// TwinCAT 3 PLC project Code
// ProgramVersion: 3.1.4026.25
// libraries:
//   ApplicationBase, * (Beckhoff Automation LLC)
//   Tc2_MC2, * (Beckhoff Automation GmbH)
//   Tc2_MC2_Camming, * (Beckhoff Automation GmbH)
//   Tc2_Standard, * (Beckhoff Automation GmbH)
//   Tc2_System, * (Beckhoff Automation GmbH)
//   XtsCore, * (Beckhoff Automation LLC)
// project tree:
//   / Godot.TcPOU, MAIN.TcPOU, PlcTask.TcTTO
//   POUs/ GodotHmi.TcPOU
//   Tests/Base/Interface/ I_SequenceTest.TcIO
//   Tests/CamBuild/ CamBuild.TcPOU, SplitCamBuild.TcPOU, ST_Camming.TcDUT
//   Tests/CamBuild/Interface/ I_CamBuildSequence.TcIO
//   Tests/CamCurveCompTest/ CamCurveComp.TcPOU, SplitCamRun.TcPOU, I_CamCurveComp.TcIO
//   Tests/ FB_XtsBallCamBuilder.TcPOU
// real-time tasks:
//   TASK PlcTask: cycle T#2ms, priority 20, ADS port 350
//   TASK XTS Task 1: cycle T#250us, priority 1, ADS port 351
//   TASK XTS AUX Task 1: cycle T#250us, priority 2, ADS port 352
//   TASK Job Task: cycle default, priority 32
// motion (NC):
//   TASK NC-Task 1: cycle T#2ms, priority 4, ADS port 501
//   TASK NC-Task 1 SVB: cycle T#10ms, priority 8, ADS port 511
//   AXIS Mover Axis 1 (id 1)
//     Dynamic: AccelerationMaximum=80000, DecelerationMaximum=80000, Acceleration=20000, Deceleration=20000, Jerk=200000
//     Velo: Maximum=4000
//     PositionAreaControl: Enable=false
//     TargetPosControl: Enable=false
//     OtherSettings: AllowMotionCmdToSlave=true, AllowMotionCmdToExtSetGenAxis=true
//     encoder EncType=28
//       EncPara: ModuloFactor=1500, ToleranceWndModuloStart=0.2, MaxCount=#xffffffff
//     drive DrvType=22
//       DrvPara: MaxCount=#xffffffff, DriveControlDWord=#x00000100
//         Analog: VeloReferenz=4200, TorqueSetpointScale=10
//         TimeComp: TaskDelayCycles=1
//     controller CtrType=1
//       CtrPara: PriorControlFactor=1
//         PosDiffControl: Range=75
//         Observer: BandWidth=20
//   AXIS Mover Axis 2 (id 2)
//     Dynamic: AccelerationMaximum=80000, DecelerationMaximum=80000, Acceleration=20000, Deceleration=20000, Jerk=200000
//     Velo: Maximum=4000
//     PositionAreaControl: Enable=false
//     TargetPosControl: Enable=false
//     OtherSettings: AllowMotionCmdToSlave=true, AllowMotionCmdToExtSetGenAxis=true
//     encoder EncType=28
//       EncPara: ModuloFactor=1500, ToleranceWndModuloStart=0.2, MaxCount=#xffffffff
//     drive DrvType=22
//       DrvPara: MaxCount=#xffffffff, DriveControlDWord=#x00000100
//         Analog: VeloReferenz=4200, TorqueSetpointScale=10
//         TimeComp: TaskDelayCycles=1
//     controller CtrType=1
//       CtrPara: PriorControlFactor=1
//         PosDiffControl: Range=50
//         Observer: BandWidth=20
//   AXIS VirtualMaster (id 3)
//     OtherSettings: AllowMotionCmdToSlave=true
//     encoder EncType=1
//       EncPara: ModuloFactor=1500
//     drive DrvType=5
//       Analog: TorqueSetpointScale=10, ScaleFactorActTorque=0.1
//       TimeComp: TaskDelayCycles=1
//     controller CtrType=1
//       CtrPara: PriorControlFactor=1
//         Observer: BandWidth=20
//   AXIS FeedAxis (id 4)
//     OtherSettings: AllowMotionCmdToSlave=true
//     encoder EncType=1
//     drive DrvType=5
//       Analog: TorqueSetpointScale=10, ScaleFactorActTorque=0.1
//       TimeComp: TaskDelayCycles=1
//     controller CtrType=1
//       CtrPara: PriorControlFactor=1
//         Observer: BandWidth=20
// I/O:
//   DEVICE Device 1 (EtherCAT), AmsNetId 192.168.1.107.2.1
//     Term 1 (EK1100) [EK1100 EtherCAT Coupler (2A E-Bus)]
//       Term 2 (EL1259) [EL1259 8Ch. Dig Input 24V/8Ch. Dig. Output 24V with Multi-Time-Stamp]
//       Term 3 (EL9227-5500) [EL9227-5500 Overcurrent protection 24V DC, 2Ch., max. 10A (sum), adjustable, extended functionalities]
//       Term 4 (EL9227-6644) [EL9227-6644 Overcurrent protection 24V DC, 2Ch., 4A/4A, extended functionalities]
//       Term 5 (EL9011) [EL9011 End Terminal]
//   DEVICE Device 2 (EtherCAT), AmsNetId 192.168.1.107.3.1
//     Term 6 (AT2102-0250) [AT2102-0250 Motormodul mit Einspeisung (B23 Steckverbinder) und NCT, 250mm, 48V]
//       Term 7 (AT2102-9250) [AT2102-9250 NCT module with feed (B23-Connector), 250mm, 48V]
//       Term 8 (AT2102-5250) [AT2102-5250 Sensor line with feed (B23-Connector) and NCT]
//     Term 9 (AT2050-0500) [AT2050-0500 Motor module, 90° clothoid, EtherCAT In, 48V]
//       Term 10 (AT2050-5500) [AT2050-5500 Sensor line 90° clothoid, EtherCAT In]
//     Term 11 (AT2050-0501) [AT2050-0501 Motor module, 90° clothoid, EtherCAT Out, 48V]
//       Term 12 (AT2050-5501) [AT2050-5501 Sensor line 90° clothoid, EtherCAT Out]
//     Term 13 (AT2100-0250) [AT2100-0250 Motormodul mit NCT, 250 mm, 48V]
//       Term 14 (AT2100-9250) [AT2100-9250 NCT module, 250mm, 48V]
//       Term 15 (AT2100-5250) [AT2100-5250 Sensor line with NCT]
//     Term 16 (AT2050-0500) [AT2050-0500 Motor module, 90° clothoid, EtherCAT In, 48V]
//       Term 17 (AT2050-5500) [AT2050-5500 Sensor line 90° clothoid, EtherCAT In]
//     Term 18 (AT2050-0501) [AT2050-0501 Motor module, 90° clothoid, EtherCAT Out, 48V]
//       Term 19 (AT2050-5501) [AT2050-5501 Sensor line 90° clothoid, EtherCAT Out]
// variable links:
//   (this object) <-> TcCOM Objects/XTS ProcessingUnit 1/Part 1/Module 1
//     Term 6 (AT2102-0250)/CC Inputs/Current actual value Ch.1 <-> Data Pointer/CurrentActualValues[0]
//     Term 6 (AT2102-0250)/CC Inputs/Current actual value Ch.10 <-> Data Pointer/CurrentActualValues[9]
//     Term 6 (AT2102-0250)/CC Inputs/Current actual value Ch.11 <-> Data Pointer/CurrentActualValues[10]
//     Term 6 (AT2102-0250)/CC Inputs/Current actual value Ch.12 <-> Data Pointer/CurrentActualValues[11]
//     Term 6 (AT2102-0250)/CC Inputs/Current actual value Ch.13 <-> Data Pointer/CurrentActualValues[12]
//     Term 6 (AT2102-0250)/CC Inputs/Current actual value Ch.14 <-> Data Pointer/CurrentActualValues[13]
//     Term 6 (AT2102-0250)/CC Inputs/Current actual value Ch.15 <-> Data Pointer/CurrentActualValues[14]
//     Term 6 (AT2102-0250)/CC Inputs/Current actual value Ch.2 <-> Data Pointer/CurrentActualValues[1]
//     Term 6 (AT2102-0250)/CC Inputs/Current actual value Ch.3 <-> Data Pointer/CurrentActualValues[2]
//     Term 6 (AT2102-0250)/CC Inputs/Current actual value Ch.4 <-> Data Pointer/CurrentActualValues[3]
//     Term 6 (AT2102-0250)/CC Inputs/Current actual value Ch.5 <-> Data Pointer/CurrentActualValues[4]
//     Term 6 (AT2102-0250)/CC Inputs/Current actual value Ch.6 <-> Data Pointer/CurrentActualValues[5]
//     Term 6 (AT2102-0250)/CC Inputs/Current actual value Ch.7 <-> Data Pointer/CurrentActualValues[6]
//     Term 6 (AT2102-0250)/CC Inputs/Current actual value Ch.8 <-> Data Pointer/CurrentActualValues[7]
//     Term 6 (AT2102-0250)/CC Inputs/Current actual value Ch.9 <-> Data Pointer/CurrentActualValues[8]
//     Term 6 (AT2102-0250)/CC Inputs/Status <-> Data Pointer/Status
//     Term 6 (AT2102-0250)/CC Outputs/Control <-> Data Pointer/Control
//     Term 6 (AT2102-0250)/CC Outputs/Current setpoint value Ch.1 <-> Data Pointer/CurrentSetpointValues[0]
//     Term 6 (AT2102-0250)/CC Outputs/Current setpoint value Ch.10 <-> Data Pointer/CurrentSetpointValues[9]
//     Term 6 (AT2102-0250)/CC Outputs/Current setpoint value Ch.11 <-> Data Pointer/CurrentSetpointValues[10]
//     Term 6 (AT2102-0250)/CC Outputs/Current setpoint value Ch.12 <-> Data Pointer/CurrentSetpointValues[11]
//     Term 6 (AT2102-0250)/CC Outputs/Current setpoint value Ch.13 <-> Data Pointer/CurrentSetpointValues[12]
//     Term 6 (AT2102-0250)/CC Outputs/Current setpoint value Ch.14 <-> Data Pointer/CurrentSetpointValues[13]
//     Term 6 (AT2102-0250)/CC Outputs/Current setpoint value Ch.15 <-> Data Pointer/CurrentSetpointValues[14]
//     Term 6 (AT2102-0250)/CC Outputs/Current setpoint value Ch.2 <-> Data Pointer/CurrentSetpointValues[1]
//     Term 6 (AT2102-0250)/CC Outputs/Current setpoint value Ch.3 <-> Data Pointer/CurrentSetpointValues[2]
//     Term 6 (AT2102-0250)/CC Outputs/Current setpoint value Ch.4 <-> Data Pointer/CurrentSetpointValues[3]
//     Term 6 (AT2102-0250)/CC Outputs/Current setpoint value Ch.5 <-> Data Pointer/CurrentSetpointValues[4]
//     Term 6 (AT2102-0250)/CC Outputs/Current setpoint value Ch.6 <-> Data Pointer/CurrentSetpointValues[5]
//     Term 6 (AT2102-0250)/CC Outputs/Current setpoint value Ch.7 <-> Data Pointer/CurrentSetpointValues[6]
//     Term 6 (AT2102-0250)/CC Outputs/Current setpoint value Ch.8 <-> Data Pointer/CurrentSetpointValues[7]
//     Term 6 (AT2102-0250)/CC Outputs/Current setpoint value Ch.9 <-> Data Pointer/CurrentSetpointValues[8]
//     Term 6 (AT2102-0250)/Term 7 (AT2102-9250)/DATA Inputs/Byte 1 <-> Data Pointer/NctInByte[1]
//     Term 6 (AT2102-0250)/Term 7 (AT2102-9250)/DATA Inputs/Byte 2 <-> Data Pointer/NctInByte[2]
//     Term 6 (AT2102-0250)/Term 7 (AT2102-9250)/DATA Inputs/Byte 3 <-> Data Pointer/NctInByte[3]
//     Term 6 (AT2102-0250)/Term 7 (AT2102-9250)/DATA Inputs/Byte 4 <-> Data Pointer/NctInByte[4]
//     Term 6 (AT2102-0250)/Term 7 (AT2102-9250)/DATA Inputs/Byte 5 <-> Data Pointer/NctInByte[5]
//     Term 6 (AT2102-0250)/Term 7 (AT2102-9250)/DATA Inputs/Byte 6 <-> Data Pointer/NctInByte[6]
//     Term 6 (AT2102-0250)/Term 7 (AT2102-9250)/DATA Inputs/Byte 7 <-> Data Pointer/NctInByte[7]
//     Term 6 (AT2102-0250)/Term 7 (AT2102-9250)/DATA Inputs/Byte 8 <-> Data Pointer/NctInByte[8]
//     Term 6 (AT2102-0250)/Term 7 (AT2102-9250)/DATA Outputs/Byte 1 <-> Data Pointer/NctOutByte[1]
//     Term 6 (AT2102-0250)/Term 7 (AT2102-9250)/DATA Outputs/Byte 2 <-> Data Pointer/NctOutByte[2]
//     Term 6 (AT2102-0250)/Term 7 (AT2102-9250)/DATA Outputs/Byte 3 <-> Data Pointer/NctOutByte[3]
//     Term 6 (AT2102-0250)/Term 7 (AT2102-9250)/DATA Outputs/Byte 4 <-> Data Pointer/NctOutByte[4]
//     Term 6 (AT2102-0250)/Term 7 (AT2102-9250)/DATA Outputs/Byte 5 <-> Data Pointer/NctOutByte[5]
//     Term 6 (AT2102-0250)/Term 7 (AT2102-9250)/DATA Outputs/Byte 6 <-> Data Pointer/NctOutByte[6]
//     Term 6 (AT2102-0250)/Term 7 (AT2102-9250)/DATA Outputs/Byte 7 <-> Data Pointer/NctOutByte[7]
//     Term 6 (AT2102-0250)/Term 7 (AT2102-9250)/DATA Outputs/Byte 8 <-> Data Pointer/NctOutByte[8]
//     Term 6 (AT2102-0250)/Term 7 (AT2102-9250)/NCT Inputs/Status <-> Data Pointer/NctStatus
//     Term 6 (AT2102-0250)/Term 7 (AT2102-9250)/NCT Outputs/Control <-> Data Pointer/NctControl
//     Term 6 (AT2102-0250)/Term 7 (AT2102-9250)/PWR Inputs Channel 1/Actual values <-> Data Pointer/NctActValues1
//     Term 6 (AT2102-0250)/Term 7 (AT2102-9250)/PWR Inputs Channel 2/Actual values <-> Data Pointer/NctActValues2
//     Term 6 (AT2102-0250)/Term 7 (AT2102-9250)/PWR Inputs Channel 1/Coil current <-> Data Pointer/NctCoilCurrent1
//     Term 6 (AT2102-0250)/Term 7 (AT2102-9250)/PWR Inputs Channel 2/Coil current <-> Data Pointer/NctCoilCurrent2
//     Term 6 (AT2102-0250)/Term 7 (AT2102-9250)/PWR Outputs Channel 1/Set values <-> Data Pointer/NctSetValues1
//     Term 6 (AT2102-0250)/Term 7 (AT2102-9250)/PWR Outputs Channel 2/Set values <-> Data Pointer/NctSetValues2
//     Term 6 (AT2102-0250)/Term 8 (AT2102-5250)/FB Inputs/Value Channel 01 <-> Data Pointer/RawPositionValues[0]
//     Term 6 (AT2102-0250)/Term 8 (AT2102-5250)/FB Inputs/Value Channel 02 <-> Data Pointer/RawPositionValues[1]
//     Term 6 (AT2102-0250)/Term 8 (AT2102-5250)/FB Inputs/Value Channel 03 <-> Data Pointer/RawPositionValues[2]
//     Term 6 (AT2102-0250)/Term 8 (AT2102-5250)/FB Inputs/Value Channel 04 <-> Data Pointer/RawPositionValues[3]
//     Term 6 (AT2102-0250)/Term 8 (AT2102-5250)/FB Inputs/Value Channel 05 <-> Data Pointer/RawPositionValues[4]
//     Term 6 (AT2102-0250)/Term 8 (AT2102-5250)/FB Inputs/Value Channel 06 <-> Data Pointer/RawPositionValues[5]
//     Term 6 (AT2102-0250)/Term 8 (AT2102-5250)/FB Inputs/Value Channel 07 <-> Data Pointer/RawPositionValues[6]
//     Term 6 (AT2102-0250)/Term 8 (AT2102-5250)/FB Inputs/Value Channel 08 <-> Data Pointer/RawPositionValues[7]
//     Term 6 (AT2102-0250)/Term 8 (AT2102-5250)/FB Inputs/Value Channel 09 <-> Data Pointer/RawPositionValues[8]
//     Term 6 (AT2102-0250)/Term 8 (AT2102-5250)/FB Inputs/Value Channel 10 <-> Data Pointer/RawPositionValues[9]
//     Term 6 (AT2102-0250)/Term 8 (AT2102-5250)/FB Inputs/Value Channel 11 <-> Data Pointer/RawPositionValues[10]
//     Term 6 (AT2102-0250)/Term 8 (AT2102-5250)/FB Inputs/Value Channel 12 <-> Data Pointer/RawPositionValues[11]
//     Term 6 (AT2102-0250)/Term 8 (AT2102-5250)/FB Inputs/Value Channel 13 <-> Data Pointer/RawPositionValues[12]
//     Term 6 (AT2102-0250)/Term 8 (AT2102-5250)/FB Inputs/Value Channel 14 <-> Data Pointer/RawPositionValues[13]
//     Term 6 (AT2102-0250)/Term 8 (AT2102-5250)/FB Inputs/Value Channel 15 <-> Data Pointer/RawPositionValues[14]
//     Term 6 (AT2102-0250)/Term 8 (AT2102-5250)/FB Inputs/Value Channel 16 <-> Data Pointer/RawPositionValues[15]
//     Term 6 (AT2102-0250)/Term 8 (AT2102-5250)/FB Inputs/Value Channel 17 <-> Data Pointer/RawPositionValues[16]
//     Term 6 (AT2102-0250)/Term 8 (AT2102-5250)/FB Inputs/Value Channel 18 <-> Data Pointer/RawPositionValues[17]
//     Term 6 (AT2102-0250)/Term 8 (AT2102-5250)/FB Inputs/Value Channel 19 <-> Data Pointer/RawPositionValues[18]
//     Term 6 (AT2102-0250)/Term 8 (AT2102-5250)/FB Inputs/Value Channel 20 <-> Data Pointer/RawPositionValues[19]
//     Term 6 (AT2102-0250)/Term 8 (AT2102-5250)/FB Inputs/Value Channel 21 <-> Data Pointer/RawPositionValues[20]
//     Term 6 (AT2102-0250)/Term 8 (AT2102-5250)/FB Inputs/Value Channel 22 <-> Data Pointer/RawPositionValues[21]
//     Term 6 (AT2102-0250)/Term 8 (AT2102-5250)/FB Inputs/Value Channel 23 <-> Data Pointer/RawPositionValues[22]
//     Term 6 (AT2102-0250)/Term 8 (AT2102-5250)/FB Inputs/Value Channel 24 <-> Data Pointer/RawPositionValues[23]
//     Term 6 (AT2102-0250)/Term 8 (AT2102-5250)/FB Inputs/Value Channel 25 <-> Data Pointer/RawPositionValues[24]
//     Term 6 (AT2102-0250)/Term 8 (AT2102-5250)/FB Inputs/Value Channel 26 <-> Data Pointer/RawPositionValues[25]
//     Term 6 (AT2102-0250)/Term 8 (AT2102-5250)/FB Inputs/Value Channel 27 <-> Data Pointer/RawPositionValues[26]
//     Term 6 (AT2102-0250)/Term 8 (AT2102-5250)/FB Inputs/Value Channel 28 <-> Data Pointer/RawPositionValues[27]
//     Term 6 (AT2102-0250)/Term 8 (AT2102-5250)/FB Inputs/Value Channel 29 <-> Data Pointer/RawPositionValues[28]
//     Term 6 (AT2102-0250)/Term 8 (AT2102-5250)/FB Inputs/Value Channel 30 <-> Data Pointer/RawPositionValues[29]
//     Term 6 (AT2102-0250)/Term 8 (AT2102-5250)/FB Inputs/Value Channel 31 <-> Data Pointer/RawPositionValues[30]
//     Term 6 (AT2102-0250)/Term 8 (AT2102-5250)/FB Inputs/Value Channel 32 <-> Data Pointer/RawPositionValues[31]
//   (this object) <-> TcCOM Objects/XTS ProcessingUnit 1/Part 1/Module 2
//     Term 9 (AT2050-0500)/CC Inputs/Current actual value Ch.1 <-> Data Pointer/CurrentActualValues[0]
//     Term 9 (AT2050-0500)/CC Inputs/Current actual value Ch.10 <-> Data Pointer/CurrentActualValues[9]
//     Term 9 (AT2050-0500)/CC Inputs/Current actual value Ch.11 <-> Data Pointer/CurrentActualValues[10]
//     Term 9 (AT2050-0500)/CC Inputs/Current actual value Ch.12 <-> Data Pointer/CurrentActualValues[11]
//     Term 9 (AT2050-0500)/CC Inputs/Current actual value Ch.13 <-> Data Pointer/CurrentActualValues[12]
//     Term 9 (AT2050-0500)/CC Inputs/Current actual value Ch.14 <-> Data Pointer/CurrentActualValues[13]
//     Term 9 (AT2050-0500)/CC Inputs/Current actual value Ch.15 <-> Data Pointer/CurrentActualValues[14]
//     Term 9 (AT2050-0500)/CC Inputs/Current actual value Ch.2 <-> Data Pointer/CurrentActualValues[1]
//     Term 9 (AT2050-0500)/CC Inputs/Current actual value Ch.3 <-> Data Pointer/CurrentActualValues[2]
//     Term 9 (AT2050-0500)/CC Inputs/Current actual value Ch.4 <-> Data Pointer/CurrentActualValues[3]
//     Term 9 (AT2050-0500)/CC Inputs/Current actual value Ch.5 <-> Data Pointer/CurrentActualValues[4]
//     Term 9 (AT2050-0500)/CC Inputs/Current actual value Ch.6 <-> Data Pointer/CurrentActualValues[5]
//     Term 9 (AT2050-0500)/CC Inputs/Current actual value Ch.7 <-> Data Pointer/CurrentActualValues[6]
//     Term 9 (AT2050-0500)/CC Inputs/Current actual value Ch.8 <-> Data Pointer/CurrentActualValues[7]
//     Term 9 (AT2050-0500)/CC Inputs/Current actual value Ch.9 <-> Data Pointer/CurrentActualValues[8]
//     Term 9 (AT2050-0500)/CC Inputs/Status <-> Data Pointer/Status
//     Term 9 (AT2050-0500)/CC Outputs/Control <-> Data Pointer/Control
//     Term 9 (AT2050-0500)/CC Outputs/Current setpoint value Ch.1 <-> Data Pointer/CurrentSetpointValues[0]
//     Term 9 (AT2050-0500)/CC Outputs/Current setpoint value Ch.10 <-> Data Pointer/CurrentSetpointValues[9]
//     Term 9 (AT2050-0500)/CC Outputs/Current setpoint value Ch.11 <-> Data Pointer/CurrentSetpointValues[10]
//     Term 9 (AT2050-0500)/CC Outputs/Current setpoint value Ch.12 <-> Data Pointer/CurrentSetpointValues[11]
//     Term 9 (AT2050-0500)/CC Outputs/Current setpoint value Ch.13 <-> Data Pointer/CurrentSetpointValues[12]
//     Term 9 (AT2050-0500)/CC Outputs/Current setpoint value Ch.14 <-> Data Pointer/CurrentSetpointValues[13]
//     Term 9 (AT2050-0500)/CC Outputs/Current setpoint value Ch.15 <-> Data Pointer/CurrentSetpointValues[14]
//     Term 9 (AT2050-0500)/CC Outputs/Current setpoint value Ch.2 <-> Data Pointer/CurrentSetpointValues[1]
//     Term 9 (AT2050-0500)/CC Outputs/Current setpoint value Ch.3 <-> Data Pointer/CurrentSetpointValues[2]
//     Term 9 (AT2050-0500)/CC Outputs/Current setpoint value Ch.4 <-> Data Pointer/CurrentSetpointValues[3]
//     Term 9 (AT2050-0500)/CC Outputs/Current setpoint value Ch.5 <-> Data Pointer/CurrentSetpointValues[4]
//     Term 9 (AT2050-0500)/CC Outputs/Current setpoint value Ch.6 <-> Data Pointer/CurrentSetpointValues[5]
//     Term 9 (AT2050-0500)/CC Outputs/Current setpoint value Ch.7 <-> Data Pointer/CurrentSetpointValues[6]
//     Term 9 (AT2050-0500)/CC Outputs/Current setpoint value Ch.8 <-> Data Pointer/CurrentSetpointValues[7]
//     Term 9 (AT2050-0500)/CC Outputs/Current setpoint value Ch.9 <-> Data Pointer/CurrentSetpointValues[8]
//     Term 9 (AT2050-0500)/Term 10 (AT2050-5500)/FB Inputs/Value Channel 01 <-> Data Pointer/RawPositionValues[0]
//     Term 9 (AT2050-0500)/Term 10 (AT2050-5500)/FB Inputs/Value Channel 02 <-> Data Pointer/RawPositionValues[1]
//     Term 9 (AT2050-0500)/Term 10 (AT2050-5500)/FB Inputs/Value Channel 03 <-> Data Pointer/RawPositionValues[2]
//     Term 9 (AT2050-0500)/Term 10 (AT2050-5500)/FB Inputs/Value Channel 04 <-> Data Pointer/RawPositionValues[3]
//     Term 9 (AT2050-0500)/Term 10 (AT2050-5500)/FB Inputs/Value Channel 05 <-> Data Pointer/RawPositionValues[4]
//     Term 9 (AT2050-0500)/Term 10 (AT2050-5500)/FB Inputs/Value Channel 06 <-> Data Pointer/RawPositionValues[5]
//     Term 9 (AT2050-0500)/Term 10 (AT2050-5500)/FB Inputs/Value Channel 07 <-> Data Pointer/RawPositionValues[6]
//     Term 9 (AT2050-0500)/Term 10 (AT2050-5500)/FB Inputs/Value Channel 08 <-> Data Pointer/RawPositionValues[7]
//     Term 9 (AT2050-0500)/Term 10 (AT2050-5500)/FB Inputs/Value Channel 09 <-> Data Pointer/RawPositionValues[8]
//     Term 9 (AT2050-0500)/Term 10 (AT2050-5500)/FB Inputs/Value Channel 10 <-> Data Pointer/RawPositionValues[9]
//     Term 9 (AT2050-0500)/Term 10 (AT2050-5500)/FB Inputs/Value Channel 11 <-> Data Pointer/RawPositionValues[10]
//     Term 9 (AT2050-0500)/Term 10 (AT2050-5500)/FB Inputs/Value Channel 12 <-> Data Pointer/RawPositionValues[11]
//     Term 9 (AT2050-0500)/Term 10 (AT2050-5500)/FB Inputs/Value Channel 13 <-> Data Pointer/RawPositionValues[12]
//     Term 9 (AT2050-0500)/Term 10 (AT2050-5500)/FB Inputs/Value Channel 14 <-> Data Pointer/RawPositionValues[13]
//     Term 9 (AT2050-0500)/Term 10 (AT2050-5500)/FB Inputs/Value Channel 15 <-> Data Pointer/RawPositionValues[14]
//     Term 9 (AT2050-0500)/Term 10 (AT2050-5500)/FB Inputs/Value Channel 16 <-> Data Pointer/RawPositionValues[15]
//     Term 9 (AT2050-0500)/Term 10 (AT2050-5500)/FB Inputs/Value Channel 17 <-> Data Pointer/RawPositionValues[16]
//     Term 9 (AT2050-0500)/Term 10 (AT2050-5500)/FB Inputs/Value Channel 18 <-> Data Pointer/RawPositionValues[17]
//     Term 9 (AT2050-0500)/Term 10 (AT2050-5500)/FB Inputs/Value Channel 19 <-> Data Pointer/RawPositionValues[18]
//     Term 9 (AT2050-0500)/Term 10 (AT2050-5500)/FB Inputs/Value Channel 20 <-> Data Pointer/RawPositionValues[19]
//     Term 9 (AT2050-0500)/Term 10 (AT2050-5500)/FB Inputs/Value Channel 21 <-> Data Pointer/RawPositionValues[20]
//     Term 9 (AT2050-0500)/Term 10 (AT2050-5500)/FB Inputs/Value Channel 22 <-> Data Pointer/RawPositionValues[21]
//     Term 9 (AT2050-0500)/Term 10 (AT2050-5500)/FB Inputs/Value Channel 23 <-> Data Pointer/RawPositionValues[22]
//     Term 9 (AT2050-0500)/Term 10 (AT2050-5500)/FB Inputs/Value Channel 24 <-> Data Pointer/RawPositionValues[23]
//     Term 9 (AT2050-0500)/Term 10 (AT2050-5500)/FB Inputs/Value Channel 25 <-> Data Pointer/RawPositionValues[24]
//     Term 9 (AT2050-0500)/Term 10 (AT2050-5500)/FB Inputs/Value Channel 26 <-> Data Pointer/RawPositionValues[25]
//     Term 9 (AT2050-0500)/Term 10 (AT2050-5500)/FB Inputs/Value Channel 27 <-> Data Pointer/RawPositionValues[26]
//     Term 9 (AT2050-0500)/Term 10 (AT2050-5500)/FB Inputs/Value Channel 28 <-> Data Pointer/RawPositionValues[27]
//     Term 9 (AT2050-0500)/Term 10 (AT2050-5500)/FB Inputs/Value Channel 29 <-> Data Pointer/RawPositionValues[28]
//     Term 9 (AT2050-0500)/Term 10 (AT2050-5500)/FB Inputs/Value Channel 30 <-> Data Pointer/RawPositionValues[29]
//     Term 9 (AT2050-0500)/Term 10 (AT2050-5500)/FB Inputs/Value Channel 31 <-> Data Pointer/RawPositionValues[30]
//     Term 9 (AT2050-0500)/Term 10 (AT2050-5500)/FB Inputs/Value Channel 32 <-> Data Pointer/RawPositionValues[31]
//   (this object) <-> TcCOM Objects/XTS ProcessingUnit 1/Part 1/Module 3
//     Term 11 (AT2050-0501)/CC Inputs/Current actual value Ch.1 <-> Data Pointer/CurrentActualValues[0]
//     Term 11 (AT2050-0501)/CC Inputs/Current actual value Ch.10 <-> Data Pointer/CurrentActualValues[9]
//     Term 11 (AT2050-0501)/CC Inputs/Current actual value Ch.11 <-> Data Pointer/CurrentActualValues[10]
//     Term 11 (AT2050-0501)/CC Inputs/Current actual value Ch.12 <-> Data Pointer/CurrentActualValues[11]
//     Term 11 (AT2050-0501)/CC Inputs/Current actual value Ch.13 <-> Data Pointer/CurrentActualValues[12]
//     Term 11 (AT2050-0501)/CC Inputs/Current actual value Ch.14 <-> Data Pointer/CurrentActualValues[13]
//     Term 11 (AT2050-0501)/CC Inputs/Current actual value Ch.15 <-> Data Pointer/CurrentActualValues[14]
//     Term 11 (AT2050-0501)/CC Inputs/Current actual value Ch.2 <-> Data Pointer/CurrentActualValues[1]
//     Term 11 (AT2050-0501)/CC Inputs/Current actual value Ch.3 <-> Data Pointer/CurrentActualValues[2]
//     Term 11 (AT2050-0501)/CC Inputs/Current actual value Ch.4 <-> Data Pointer/CurrentActualValues[3]
//     Term 11 (AT2050-0501)/CC Inputs/Current actual value Ch.5 <-> Data Pointer/CurrentActualValues[4]
//     Term 11 (AT2050-0501)/CC Inputs/Current actual value Ch.6 <-> Data Pointer/CurrentActualValues[5]
//     Term 11 (AT2050-0501)/CC Inputs/Current actual value Ch.7 <-> Data Pointer/CurrentActualValues[6]
//     Term 11 (AT2050-0501)/CC Inputs/Current actual value Ch.8 <-> Data Pointer/CurrentActualValues[7]
//     Term 11 (AT2050-0501)/CC Inputs/Current actual value Ch.9 <-> Data Pointer/CurrentActualValues[8]
//     Term 11 (AT2050-0501)/CC Inputs/Status <-> Data Pointer/Status
//     Term 11 (AT2050-0501)/CC Outputs/Control <-> Data Pointer/Control
//     Term 11 (AT2050-0501)/CC Outputs/Current setpoint value Ch.1 <-> Data Pointer/CurrentSetpointValues[0]
//     Term 11 (AT2050-0501)/CC Outputs/Current setpoint value Ch.10 <-> Data Pointer/CurrentSetpointValues[9]
//     Term 11 (AT2050-0501)/CC Outputs/Current setpoint value Ch.11 <-> Data Pointer/CurrentSetpointValues[10]
//     Term 11 (AT2050-0501)/CC Outputs/Current setpoint value Ch.12 <-> Data Pointer/CurrentSetpointValues[11]
//     Term 11 (AT2050-0501)/CC Outputs/Current setpoint value Ch.13 <-> Data Pointer/CurrentSetpointValues[12]
//     Term 11 (AT2050-0501)/CC Outputs/Current setpoint value Ch.14 <-> Data Pointer/CurrentSetpointValues[13]
//     Term 11 (AT2050-0501)/CC Outputs/Current setpoint value Ch.15 <-> Data Pointer/CurrentSetpointValues[14]
//     Term 11 (AT2050-0501)/CC Outputs/Current setpoint value Ch.2 <-> Data Pointer/CurrentSetpointValues[1]
//     Term 11 (AT2050-0501)/CC Outputs/Current setpoint value Ch.3 <-> Data Pointer/CurrentSetpointValues[2]
//     Term 11 (AT2050-0501)/CC Outputs/Current setpoint value Ch.4 <-> Data Pointer/CurrentSetpointValues[3]
//     Term 11 (AT2050-0501)/CC Outputs/Current setpoint value Ch.5 <-> Data Pointer/CurrentSetpointValues[4]
//     Term 11 (AT2050-0501)/CC Outputs/Current setpoint value Ch.6 <-> Data Pointer/CurrentSetpointValues[5]
//     Term 11 (AT2050-0501)/CC Outputs/Current setpoint value Ch.7 <-> Data Pointer/CurrentSetpointValues[6]
//     Term 11 (AT2050-0501)/CC Outputs/Current setpoint value Ch.8 <-> Data Pointer/CurrentSetpointValues[7]
//     Term 11 (AT2050-0501)/CC Outputs/Current setpoint value Ch.9 <-> Data Pointer/CurrentSetpointValues[8]
//     Term 11 (AT2050-0501)/Term 12 (AT2050-5501)/FB Inputs/Value Channel 01 <-> Data Pointer/RawPositionValues[0]
//     Term 11 (AT2050-0501)/Term 12 (AT2050-5501)/FB Inputs/Value Channel 02 <-> Data Pointer/RawPositionValues[1]
//     Term 11 (AT2050-0501)/Term 12 (AT2050-5501)/FB Inputs/Value Channel 03 <-> Data Pointer/RawPositionValues[2]
//     Term 11 (AT2050-0501)/Term 12 (AT2050-5501)/FB Inputs/Value Channel 04 <-> Data Pointer/RawPositionValues[3]
//     Term 11 (AT2050-0501)/Term 12 (AT2050-5501)/FB Inputs/Value Channel 05 <-> Data Pointer/RawPositionValues[4]
//     Term 11 (AT2050-0501)/Term 12 (AT2050-5501)/FB Inputs/Value Channel 06 <-> Data Pointer/RawPositionValues[5]
//     Term 11 (AT2050-0501)/Term 12 (AT2050-5501)/FB Inputs/Value Channel 07 <-> Data Pointer/RawPositionValues[6]
//     Term 11 (AT2050-0501)/Term 12 (AT2050-5501)/FB Inputs/Value Channel 08 <-> Data Pointer/RawPositionValues[7]
//     Term 11 (AT2050-0501)/Term 12 (AT2050-5501)/FB Inputs/Value Channel 09 <-> Data Pointer/RawPositionValues[8]
//     Term 11 (AT2050-0501)/Term 12 (AT2050-5501)/FB Inputs/Value Channel 10 <-> Data Pointer/RawPositionValues[9]
//     Term 11 (AT2050-0501)/Term 12 (AT2050-5501)/FB Inputs/Value Channel 11 <-> Data Pointer/RawPositionValues[10]
//     Term 11 (AT2050-0501)/Term 12 (AT2050-5501)/FB Inputs/Value Channel 12 <-> Data Pointer/RawPositionValues[11]
//     Term 11 (AT2050-0501)/Term 12 (AT2050-5501)/FB Inputs/Value Channel 13 <-> Data Pointer/RawPositionValues[12]
//     Term 11 (AT2050-0501)/Term 12 (AT2050-5501)/FB Inputs/Value Channel 14 <-> Data Pointer/RawPositionValues[13]
//     Term 11 (AT2050-0501)/Term 12 (AT2050-5501)/FB Inputs/Value Channel 15 <-> Data Pointer/RawPositionValues[14]
//     Term 11 (AT2050-0501)/Term 12 (AT2050-5501)/FB Inputs/Value Channel 16 <-> Data Pointer/RawPositionValues[15]
//     Term 11 (AT2050-0501)/Term 12 (AT2050-5501)/FB Inputs/Value Channel 17 <-> Data Pointer/RawPositionValues[16]
//     Term 11 (AT2050-0501)/Term 12 (AT2050-5501)/FB Inputs/Value Channel 18 <-> Data Pointer/RawPositionValues[17]
//     Term 11 (AT2050-0501)/Term 12 (AT2050-5501)/FB Inputs/Value Channel 19 <-> Data Pointer/RawPositionValues[18]
//     Term 11 (AT2050-0501)/Term 12 (AT2050-5501)/FB Inputs/Value Channel 20 <-> Data Pointer/RawPositionValues[19]
//     Term 11 (AT2050-0501)/Term 12 (AT2050-5501)/FB Inputs/Value Channel 21 <-> Data Pointer/RawPositionValues[20]
//     Term 11 (AT2050-0501)/Term 12 (AT2050-5501)/FB Inputs/Value Channel 22 <-> Data Pointer/RawPositionValues[21]
//     Term 11 (AT2050-0501)/Term 12 (AT2050-5501)/FB Inputs/Value Channel 23 <-> Data Pointer/RawPositionValues[22]
//     Term 11 (AT2050-0501)/Term 12 (AT2050-5501)/FB Inputs/Value Channel 24 <-> Data Pointer/RawPositionValues[23]
//     Term 11 (AT2050-0501)/Term 12 (AT2050-5501)/FB Inputs/Value Channel 25 <-> Data Pointer/RawPositionValues[24]
//     Term 11 (AT2050-0501)/Term 12 (AT2050-5501)/FB Inputs/Value Channel 26 <-> Data Pointer/RawPositionValues[25]
//     Term 11 (AT2050-0501)/Term 12 (AT2050-5501)/FB Inputs/Value Channel 27 <-> Data Pointer/RawPositionValues[26]
//     Term 11 (AT2050-0501)/Term 12 (AT2050-5501)/FB Inputs/Value Channel 28 <-> Data Pointer/RawPositionValues[27]
//     Term 11 (AT2050-0501)/Term 12 (AT2050-5501)/FB Inputs/Value Channel 29 <-> Data Pointer/RawPositionValues[28]
//     Term 11 (AT2050-0501)/Term 12 (AT2050-5501)/FB Inputs/Value Channel 30 <-> Data Pointer/RawPositionValues[29]
//     Term 11 (AT2050-0501)/Term 12 (AT2050-5501)/FB Inputs/Value Channel 31 <-> Data Pointer/RawPositionValues[30]
//     Term 11 (AT2050-0501)/Term 12 (AT2050-5501)/FB Inputs/Value Channel 32 <-> Data Pointer/RawPositionValues[31]
//   (this object) <-> TcCOM Objects/XTS ProcessingUnit 1/Part 1/Module 4
//     Term 13 (AT2100-0250)/CC Inputs/Current actual value Ch.1 <-> Data Pointer/CurrentActualValues[0]
//     Term 13 (AT2100-0250)/CC Inputs/Current actual value Ch.10 <-> Data Pointer/CurrentActualValues[9]
//     Term 13 (AT2100-0250)/CC Inputs/Current actual value Ch.11 <-> Data Pointer/CurrentActualValues[10]
//     Term 13 (AT2100-0250)/CC Inputs/Current actual value Ch.12 <-> Data Pointer/CurrentActualValues[11]
//     Term 13 (AT2100-0250)/CC Inputs/Current actual value Ch.13 <-> Data Pointer/CurrentActualValues[12]
//     Term 13 (AT2100-0250)/CC Inputs/Current actual value Ch.14 <-> Data Pointer/CurrentActualValues[13]
//     Term 13 (AT2100-0250)/CC Inputs/Current actual value Ch.15 <-> Data Pointer/CurrentActualValues[14]
//     Term 13 (AT2100-0250)/CC Inputs/Current actual value Ch.2 <-> Data Pointer/CurrentActualValues[1]
//     Term 13 (AT2100-0250)/CC Inputs/Current actual value Ch.3 <-> Data Pointer/CurrentActualValues[2]
//     Term 13 (AT2100-0250)/CC Inputs/Current actual value Ch.4 <-> Data Pointer/CurrentActualValues[3]
//     Term 13 (AT2100-0250)/CC Inputs/Current actual value Ch.5 <-> Data Pointer/CurrentActualValues[4]
//     Term 13 (AT2100-0250)/CC Inputs/Current actual value Ch.6 <-> Data Pointer/CurrentActualValues[5]
//     Term 13 (AT2100-0250)/CC Inputs/Current actual value Ch.7 <-> Data Pointer/CurrentActualValues[6]
//     Term 13 (AT2100-0250)/CC Inputs/Current actual value Ch.8 <-> Data Pointer/CurrentActualValues[7]
//     Term 13 (AT2100-0250)/CC Inputs/Current actual value Ch.9 <-> Data Pointer/CurrentActualValues[8]
//     Term 13 (AT2100-0250)/CC Inputs/Status <-> Data Pointer/Status
//     Term 13 (AT2100-0250)/CC Outputs/Control <-> Data Pointer/Control
//     Term 13 (AT2100-0250)/CC Outputs/Current setpoint value Ch.1 <-> Data Pointer/CurrentSetpointValues[0]
//     Term 13 (AT2100-0250)/CC Outputs/Current setpoint value Ch.10 <-> Data Pointer/CurrentSetpointValues[9]
//     Term 13 (AT2100-0250)/CC Outputs/Current setpoint value Ch.11 <-> Data Pointer/CurrentSetpointValues[10]
//     Term 13 (AT2100-0250)/CC Outputs/Current setpoint value Ch.12 <-> Data Pointer/CurrentSetpointValues[11]
//     Term 13 (AT2100-0250)/CC Outputs/Current setpoint value Ch.13 <-> Data Pointer/CurrentSetpointValues[12]
//     Term 13 (AT2100-0250)/CC Outputs/Current setpoint value Ch.14 <-> Data Pointer/CurrentSetpointValues[13]
//     Term 13 (AT2100-0250)/CC Outputs/Current setpoint value Ch.15 <-> Data Pointer/CurrentSetpointValues[14]
//     Term 13 (AT2100-0250)/CC Outputs/Current setpoint value Ch.2 <-> Data Pointer/CurrentSetpointValues[1]
//     Term 13 (AT2100-0250)/CC Outputs/Current setpoint value Ch.3 <-> Data Pointer/CurrentSetpointValues[2]
//     Term 13 (AT2100-0250)/CC Outputs/Current setpoint value Ch.4 <-> Data Pointer/CurrentSetpointValues[3]
//     Term 13 (AT2100-0250)/CC Outputs/Current setpoint value Ch.5 <-> Data Pointer/CurrentSetpointValues[4]
//     Term 13 (AT2100-0250)/CC Outputs/Current setpoint value Ch.6 <-> Data Pointer/CurrentSetpointValues[5]
//     Term 13 (AT2100-0250)/CC Outputs/Current setpoint value Ch.7 <-> Data Pointer/CurrentSetpointValues[6]
//     Term 13 (AT2100-0250)/CC Outputs/Current setpoint value Ch.8 <-> Data Pointer/CurrentSetpointValues[7]
//     Term 13 (AT2100-0250)/CC Outputs/Current setpoint value Ch.9 <-> Data Pointer/CurrentSetpointValues[8]
//     Term 13 (AT2100-0250)/Term 14 (AT2100-9250)/DATA Inputs/Byte 1 <-> Data Pointer/NctInByte[1]
//     Term 13 (AT2100-0250)/Term 14 (AT2100-9250)/DATA Inputs/Byte 2 <-> Data Pointer/NctInByte[2]
//     Term 13 (AT2100-0250)/Term 14 (AT2100-9250)/DATA Inputs/Byte 3 <-> Data Pointer/NctInByte[3]
//     Term 13 (AT2100-0250)/Term 14 (AT2100-9250)/DATA Inputs/Byte 4 <-> Data Pointer/NctInByte[4]
//     Term 13 (AT2100-0250)/Term 14 (AT2100-9250)/DATA Inputs/Byte 5 <-> Data Pointer/NctInByte[5]
//     Term 13 (AT2100-0250)/Term 14 (AT2100-9250)/DATA Inputs/Byte 6 <-> Data Pointer/NctInByte[6]
//     Term 13 (AT2100-0250)/Term 14 (AT2100-9250)/DATA Inputs/Byte 7 <-> Data Pointer/NctInByte[7]
//     Term 13 (AT2100-0250)/Term 14 (AT2100-9250)/DATA Inputs/Byte 8 <-> Data Pointer/NctInByte[8]
//     Term 13 (AT2100-0250)/Term 14 (AT2100-9250)/DATA Outputs/Byte 1 <-> Data Pointer/NctOutByte[1]
//     Term 13 (AT2100-0250)/Term 14 (AT2100-9250)/DATA Outputs/Byte 2 <-> Data Pointer/NctOutByte[2]
//     Term 13 (AT2100-0250)/Term 14 (AT2100-9250)/DATA Outputs/Byte 3 <-> Data Pointer/NctOutByte[3]
//     Term 13 (AT2100-0250)/Term 14 (AT2100-9250)/DATA Outputs/Byte 4 <-> Data Pointer/NctOutByte[4]
//     Term 13 (AT2100-0250)/Term 14 (AT2100-9250)/DATA Outputs/Byte 5 <-> Data Pointer/NctOutByte[5]
//     Term 13 (AT2100-0250)/Term 14 (AT2100-9250)/DATA Outputs/Byte 6 <-> Data Pointer/NctOutByte[6]
//     Term 13 (AT2100-0250)/Term 14 (AT2100-9250)/DATA Outputs/Byte 7 <-> Data Pointer/NctOutByte[7]
//     Term 13 (AT2100-0250)/Term 14 (AT2100-9250)/DATA Outputs/Byte 8 <-> Data Pointer/NctOutByte[8]
//     Term 13 (AT2100-0250)/Term 14 (AT2100-9250)/NCT Inputs/Status <-> Data Pointer/NctStatus
//     Term 13 (AT2100-0250)/Term 14 (AT2100-9250)/NCT Outputs/Control <-> Data Pointer/NctControl
//     Term 13 (AT2100-0250)/Term 14 (AT2100-9250)/PWR Inputs Channel 1/Actual values <-> Data Pointer/NctActValues1
//     Term 13 (AT2100-0250)/Term 14 (AT2100-9250)/PWR Inputs Channel 2/Actual values <-> Data Pointer/NctActValues2
//     Term 13 (AT2100-0250)/Term 14 (AT2100-9250)/PWR Inputs Channel 1/Coil current <-> Data Pointer/NctCoilCurrent1
//     Term 13 (AT2100-0250)/Term 14 (AT2100-9250)/PWR Inputs Channel 2/Coil current <-> Data Pointer/NctCoilCurrent2
//     Term 13 (AT2100-0250)/Term 14 (AT2100-9250)/PWR Outputs Channel 1/Set values <-> Data Pointer/NctSetValues1
//     Term 13 (AT2100-0250)/Term 14 (AT2100-9250)/PWR Outputs Channel 2/Set values <-> Data Pointer/NctSetValues2
//     Term 13 (AT2100-0250)/Term 15 (AT2100-5250)/FB Inputs/Value Channel 01 <-> Data Pointer/RawPositionValues[0]
//     Term 13 (AT2100-0250)/Term 15 (AT2100-5250)/FB Inputs/Value Channel 02 <-> Data Pointer/RawPositionValues[1]
//     Term 13 (AT2100-0250)/Term 15 (AT2100-5250)/FB Inputs/Value Channel 03 <-> Data Pointer/RawPositionValues[2]
//     Term 13 (AT2100-0250)/Term 15 (AT2100-5250)/FB Inputs/Value Channel 04 <-> Data Pointer/RawPositionValues[3]
//     Term 13 (AT2100-0250)/Term 15 (AT2100-5250)/FB Inputs/Value Channel 05 <-> Data Pointer/RawPositionValues[4]
//     Term 13 (AT2100-0250)/Term 15 (AT2100-5250)/FB Inputs/Value Channel 06 <-> Data Pointer/RawPositionValues[5]
//     Term 13 (AT2100-0250)/Term 15 (AT2100-5250)/FB Inputs/Value Channel 07 <-> Data Pointer/RawPositionValues[6]
//     Term 13 (AT2100-0250)/Term 15 (AT2100-5250)/FB Inputs/Value Channel 08 <-> Data Pointer/RawPositionValues[7]
//     Term 13 (AT2100-0250)/Term 15 (AT2100-5250)/FB Inputs/Value Channel 09 <-> Data Pointer/RawPositionValues[8]
//     Term 13 (AT2100-0250)/Term 15 (AT2100-5250)/FB Inputs/Value Channel 10 <-> Data Pointer/RawPositionValues[9]
//     Term 13 (AT2100-0250)/Term 15 (AT2100-5250)/FB Inputs/Value Channel 11 <-> Data Pointer/RawPositionValues[10]
//     Term 13 (AT2100-0250)/Term 15 (AT2100-5250)/FB Inputs/Value Channel 12 <-> Data Pointer/RawPositionValues[11]
//     Term 13 (AT2100-0250)/Term 15 (AT2100-5250)/FB Inputs/Value Channel 13 <-> Data Pointer/RawPositionValues[12]
//     Term 13 (AT2100-0250)/Term 15 (AT2100-5250)/FB Inputs/Value Channel 14 <-> Data Pointer/RawPositionValues[13]
//     Term 13 (AT2100-0250)/Term 15 (AT2100-5250)/FB Inputs/Value Channel 15 <-> Data Pointer/RawPositionValues[14]
//     Term 13 (AT2100-0250)/Term 15 (AT2100-5250)/FB Inputs/Value Channel 16 <-> Data Pointer/RawPositionValues[15]
//     Term 13 (AT2100-0250)/Term 15 (AT2100-5250)/FB Inputs/Value Channel 17 <-> Data Pointer/RawPositionValues[16]
//     Term 13 (AT2100-0250)/Term 15 (AT2100-5250)/FB Inputs/Value Channel 18 <-> Data Pointer/RawPositionValues[17]
//     Term 13 (AT2100-0250)/Term 15 (AT2100-5250)/FB Inputs/Value Channel 19 <-> Data Pointer/RawPositionValues[18]
//     Term 13 (AT2100-0250)/Term 15 (AT2100-5250)/FB Inputs/Value Channel 20 <-> Data Pointer/RawPositionValues[19]
//     Term 13 (AT2100-0250)/Term 15 (AT2100-5250)/FB Inputs/Value Channel 21 <-> Data Pointer/RawPositionValues[20]
//     Term 13 (AT2100-0250)/Term 15 (AT2100-5250)/FB Inputs/Value Channel 22 <-> Data Pointer/RawPositionValues[21]
//     Term 13 (AT2100-0250)/Term 15 (AT2100-5250)/FB Inputs/Value Channel 23 <-> Data Pointer/RawPositionValues[22]
//     Term 13 (AT2100-0250)/Term 15 (AT2100-5250)/FB Inputs/Value Channel 24 <-> Data Pointer/RawPositionValues[23]
//     Term 13 (AT2100-0250)/Term 15 (AT2100-5250)/FB Inputs/Value Channel 25 <-> Data Pointer/RawPositionValues[24]
//     Term 13 (AT2100-0250)/Term 15 (AT2100-5250)/FB Inputs/Value Channel 26 <-> Data Pointer/RawPositionValues[25]
//     Term 13 (AT2100-0250)/Term 15 (AT2100-5250)/FB Inputs/Value Channel 27 <-> Data Pointer/RawPositionValues[26]
//     Term 13 (AT2100-0250)/Term 15 (AT2100-5250)/FB Inputs/Value Channel 28 <-> Data Pointer/RawPositionValues[27]
//     Term 13 (AT2100-0250)/Term 15 (AT2100-5250)/FB Inputs/Value Channel 29 <-> Data Pointer/RawPositionValues[28]
//     Term 13 (AT2100-0250)/Term 15 (AT2100-5250)/FB Inputs/Value Channel 30 <-> Data Pointer/RawPositionValues[29]
//     Term 13 (AT2100-0250)/Term 15 (AT2100-5250)/FB Inputs/Value Channel 31 <-> Data Pointer/RawPositionValues[30]
//     Term 13 (AT2100-0250)/Term 15 (AT2100-5250)/FB Inputs/Value Channel 32 <-> Data Pointer/RawPositionValues[31]
//   (this object) <-> TcCOM Objects/XTS ProcessingUnit 1/Part 1/Module 5
//     Term 16 (AT2050-0500)/CC Inputs/Current actual value Ch.1 <-> Data Pointer/CurrentActualValues[0]
//     Term 16 (AT2050-0500)/CC Inputs/Current actual value Ch.10 <-> Data Pointer/CurrentActualValues[9]
//     Term 16 (AT2050-0500)/CC Inputs/Current actual value Ch.11 <-> Data Pointer/CurrentActualValues[10]
//     Term 16 (AT2050-0500)/CC Inputs/Current actual value Ch.12 <-> Data Pointer/CurrentActualValues[11]
//     Term 16 (AT2050-0500)/CC Inputs/Current actual value Ch.13 <-> Data Pointer/CurrentActualValues[12]
//     Term 16 (AT2050-0500)/CC Inputs/Current actual value Ch.14 <-> Data Pointer/CurrentActualValues[13]
//     Term 16 (AT2050-0500)/CC Inputs/Current actual value Ch.15 <-> Data Pointer/CurrentActualValues[14]
//     Term 16 (AT2050-0500)/CC Inputs/Current actual value Ch.2 <-> Data Pointer/CurrentActualValues[1]
//     Term 16 (AT2050-0500)/CC Inputs/Current actual value Ch.3 <-> Data Pointer/CurrentActualValues[2]
//     Term 16 (AT2050-0500)/CC Inputs/Current actual value Ch.4 <-> Data Pointer/CurrentActualValues[3]
//     Term 16 (AT2050-0500)/CC Inputs/Current actual value Ch.5 <-> Data Pointer/CurrentActualValues[4]
//     Term 16 (AT2050-0500)/CC Inputs/Current actual value Ch.6 <-> Data Pointer/CurrentActualValues[5]
//     Term 16 (AT2050-0500)/CC Inputs/Current actual value Ch.7 <-> Data Pointer/CurrentActualValues[6]
//     Term 16 (AT2050-0500)/CC Inputs/Current actual value Ch.8 <-> Data Pointer/CurrentActualValues[7]
//     Term 16 (AT2050-0500)/CC Inputs/Current actual value Ch.9 <-> Data Pointer/CurrentActualValues[8]
//     Term 16 (AT2050-0500)/CC Inputs/Status <-> Data Pointer/Status
//     Term 16 (AT2050-0500)/CC Outputs/Control <-> Data Pointer/Control
//     Term 16 (AT2050-0500)/CC Outputs/Current setpoint value Ch.1 <-> Data Pointer/CurrentSetpointValues[0]
//     Term 16 (AT2050-0500)/CC Outputs/Current setpoint value Ch.10 <-> Data Pointer/CurrentSetpointValues[9]
//     Term 16 (AT2050-0500)/CC Outputs/Current setpoint value Ch.11 <-> Data Pointer/CurrentSetpointValues[10]
//     Term 16 (AT2050-0500)/CC Outputs/Current setpoint value Ch.12 <-> Data Pointer/CurrentSetpointValues[11]
//     Term 16 (AT2050-0500)/CC Outputs/Current setpoint value Ch.13 <-> Data Pointer/CurrentSetpointValues[12]
//     Term 16 (AT2050-0500)/CC Outputs/Current setpoint value Ch.14 <-> Data Pointer/CurrentSetpointValues[13]
//     Term 16 (AT2050-0500)/CC Outputs/Current setpoint value Ch.15 <-> Data Pointer/CurrentSetpointValues[14]
//     Term 16 (AT2050-0500)/CC Outputs/Current setpoint value Ch.2 <-> Data Pointer/CurrentSetpointValues[1]
//     Term 16 (AT2050-0500)/CC Outputs/Current setpoint value Ch.3 <-> Data Pointer/CurrentSetpointValues[2]
//     Term 16 (AT2050-0500)/CC Outputs/Current setpoint value Ch.4 <-> Data Pointer/CurrentSetpointValues[3]
//     Term 16 (AT2050-0500)/CC Outputs/Current setpoint value Ch.5 <-> Data Pointer/CurrentSetpointValues[4]
//     Term 16 (AT2050-0500)/CC Outputs/Current setpoint value Ch.6 <-> Data Pointer/CurrentSetpointValues[5]
//     Term 16 (AT2050-0500)/CC Outputs/Current setpoint value Ch.7 <-> Data Pointer/CurrentSetpointValues[6]
//     Term 16 (AT2050-0500)/CC Outputs/Current setpoint value Ch.8 <-> Data Pointer/CurrentSetpointValues[7]
//     Term 16 (AT2050-0500)/CC Outputs/Current setpoint value Ch.9 <-> Data Pointer/CurrentSetpointValues[8]
//     Term 16 (AT2050-0500)/Term 17 (AT2050-5500)/FB Inputs/Value Channel 01 <-> Data Pointer/RawPositionValues[0]
//     Term 16 (AT2050-0500)/Term 17 (AT2050-5500)/FB Inputs/Value Channel 02 <-> Data Pointer/RawPositionValues[1]
//     Term 16 (AT2050-0500)/Term 17 (AT2050-5500)/FB Inputs/Value Channel 03 <-> Data Pointer/RawPositionValues[2]
//     Term 16 (AT2050-0500)/Term 17 (AT2050-5500)/FB Inputs/Value Channel 04 <-> Data Pointer/RawPositionValues[3]
//     Term 16 (AT2050-0500)/Term 17 (AT2050-5500)/FB Inputs/Value Channel 05 <-> Data Pointer/RawPositionValues[4]
//     Term 16 (AT2050-0500)/Term 17 (AT2050-5500)/FB Inputs/Value Channel 06 <-> Data Pointer/RawPositionValues[5]
//     Term 16 (AT2050-0500)/Term 17 (AT2050-5500)/FB Inputs/Value Channel 07 <-> Data Pointer/RawPositionValues[6]
//     Term 16 (AT2050-0500)/Term 17 (AT2050-5500)/FB Inputs/Value Channel 08 <-> Data Pointer/RawPositionValues[7]
//     Term 16 (AT2050-0500)/Term 17 (AT2050-5500)/FB Inputs/Value Channel 09 <-> Data Pointer/RawPositionValues[8]
//     Term 16 (AT2050-0500)/Term 17 (AT2050-5500)/FB Inputs/Value Channel 10 <-> Data Pointer/RawPositionValues[9]
//     Term 16 (AT2050-0500)/Term 17 (AT2050-5500)/FB Inputs/Value Channel 11 <-> Data Pointer/RawPositionValues[10]
//     Term 16 (AT2050-0500)/Term 17 (AT2050-5500)/FB Inputs/Value Channel 12 <-> Data Pointer/RawPositionValues[11]
//     Term 16 (AT2050-0500)/Term 17 (AT2050-5500)/FB Inputs/Value Channel 13 <-> Data Pointer/RawPositionValues[12]
//     Term 16 (AT2050-0500)/Term 17 (AT2050-5500)/FB Inputs/Value Channel 14 <-> Data Pointer/RawPositionValues[13]
//     Term 16 (AT2050-0500)/Term 17 (AT2050-5500)/FB Inputs/Value Channel 15 <-> Data Pointer/RawPositionValues[14]
//     Term 16 (AT2050-0500)/Term 17 (AT2050-5500)/FB Inputs/Value Channel 16 <-> Data Pointer/RawPositionValues[15]
//     Term 16 (AT2050-0500)/Term 17 (AT2050-5500)/FB Inputs/Value Channel 17 <-> Data Pointer/RawPositionValues[16]
//     Term 16 (AT2050-0500)/Term 17 (AT2050-5500)/FB Inputs/Value Channel 18 <-> Data Pointer/RawPositionValues[17]
//     Term 16 (AT2050-0500)/Term 17 (AT2050-5500)/FB Inputs/Value Channel 19 <-> Data Pointer/RawPositionValues[18]
//     Term 16 (AT2050-0500)/Term 17 (AT2050-5500)/FB Inputs/Value Channel 20 <-> Data Pointer/RawPositionValues[19]
//     Term 16 (AT2050-0500)/Term 17 (AT2050-5500)/FB Inputs/Value Channel 21 <-> Data Pointer/RawPositionValues[20]
//     Term 16 (AT2050-0500)/Term 17 (AT2050-5500)/FB Inputs/Value Channel 22 <-> Data Pointer/RawPositionValues[21]
//     Term 16 (AT2050-0500)/Term 17 (AT2050-5500)/FB Inputs/Value Channel 23 <-> Data Pointer/RawPositionValues[22]
//     Term 16 (AT2050-0500)/Term 17 (AT2050-5500)/FB Inputs/Value Channel 24 <-> Data Pointer/RawPositionValues[23]
//     Term 16 (AT2050-0500)/Term 17 (AT2050-5500)/FB Inputs/Value Channel 25 <-> Data Pointer/RawPositionValues[24]
//     Term 16 (AT2050-0500)/Term 17 (AT2050-5500)/FB Inputs/Value Channel 26 <-> Data Pointer/RawPositionValues[25]
//     Term 16 (AT2050-0500)/Term 17 (AT2050-5500)/FB Inputs/Value Channel 27 <-> Data Pointer/RawPositionValues[26]
//     Term 16 (AT2050-0500)/Term 17 (AT2050-5500)/FB Inputs/Value Channel 28 <-> Data Pointer/RawPositionValues[27]
//     Term 16 (AT2050-0500)/Term 17 (AT2050-5500)/FB Inputs/Value Channel 29 <-> Data Pointer/RawPositionValues[28]
//     Term 16 (AT2050-0500)/Term 17 (AT2050-5500)/FB Inputs/Value Channel 30 <-> Data Pointer/RawPositionValues[29]
//     Term 16 (AT2050-0500)/Term 17 (AT2050-5500)/FB Inputs/Value Channel 31 <-> Data Pointer/RawPositionValues[30]
//     Term 16 (AT2050-0500)/Term 17 (AT2050-5500)/FB Inputs/Value Channel 32 <-> Data Pointer/RawPositionValues[31]
//   (this object) <-> TcCOM Objects/XTS ProcessingUnit 1/Part 1/Module 6
//     Term 18 (AT2050-0501)/CC Inputs/Current actual value Ch.1 <-> Data Pointer/CurrentActualValues[0]
//     Term 18 (AT2050-0501)/CC Inputs/Current actual value Ch.10 <-> Data Pointer/CurrentActualValues[9]
//     Term 18 (AT2050-0501)/CC Inputs/Current actual value Ch.11 <-> Data Pointer/CurrentActualValues[10]
//     Term 18 (AT2050-0501)/CC Inputs/Current actual value Ch.12 <-> Data Pointer/CurrentActualValues[11]
//     Term 18 (AT2050-0501)/CC Inputs/Current actual value Ch.13 <-> Data Pointer/CurrentActualValues[12]
//     Term 18 (AT2050-0501)/CC Inputs/Current actual value Ch.14 <-> Data Pointer/CurrentActualValues[13]
//     Term 18 (AT2050-0501)/CC Inputs/Current actual value Ch.15 <-> Data Pointer/CurrentActualValues[14]
//     Term 18 (AT2050-0501)/CC Inputs/Current actual value Ch.2 <-> Data Pointer/CurrentActualValues[1]
//     Term 18 (AT2050-0501)/CC Inputs/Current actual value Ch.3 <-> Data Pointer/CurrentActualValues[2]
//     Term 18 (AT2050-0501)/CC Inputs/Current actual value Ch.4 <-> Data Pointer/CurrentActualValues[3]
//     Term 18 (AT2050-0501)/CC Inputs/Current actual value Ch.5 <-> Data Pointer/CurrentActualValues[4]
//     Term 18 (AT2050-0501)/CC Inputs/Current actual value Ch.6 <-> Data Pointer/CurrentActualValues[5]
//     Term 18 (AT2050-0501)/CC Inputs/Current actual value Ch.7 <-> Data Pointer/CurrentActualValues[6]
//     Term 18 (AT2050-0501)/CC Inputs/Current actual value Ch.8 <-> Data Pointer/CurrentActualValues[7]
//     Term 18 (AT2050-0501)/CC Inputs/Current actual value Ch.9 <-> Data Pointer/CurrentActualValues[8]
//     Term 18 (AT2050-0501)/CC Inputs/Status <-> Data Pointer/Status
//     Term 18 (AT2050-0501)/CC Outputs/Control <-> Data Pointer/Control
//     Term 18 (AT2050-0501)/CC Outputs/Current setpoint value Ch.1 <-> Data Pointer/CurrentSetpointValues[0]
//     Term 18 (AT2050-0501)/CC Outputs/Current setpoint value Ch.10 <-> Data Pointer/CurrentSetpointValues[9]
//     Term 18 (AT2050-0501)/CC Outputs/Current setpoint value Ch.11 <-> Data Pointer/CurrentSetpointValues[10]
//     Term 18 (AT2050-0501)/CC Outputs/Current setpoint value Ch.12 <-> Data Pointer/CurrentSetpointValues[11]
//     Term 18 (AT2050-0501)/CC Outputs/Current setpoint value Ch.13 <-> Data Pointer/CurrentSetpointValues[12]
//     Term 18 (AT2050-0501)/CC Outputs/Current setpoint value Ch.14 <-> Data Pointer/CurrentSetpointValues[13]
//     Term 18 (AT2050-0501)/CC Outputs/Current setpoint value Ch.15 <-> Data Pointer/CurrentSetpointValues[14]
//     Term 18 (AT2050-0501)/CC Outputs/Current setpoint value Ch.2 <-> Data Pointer/CurrentSetpointValues[1]
//     Term 18 (AT2050-0501)/CC Outputs/Current setpoint value Ch.3 <-> Data Pointer/CurrentSetpointValues[2]
//     Term 18 (AT2050-0501)/CC Outputs/Current setpoint value Ch.4 <-> Data Pointer/CurrentSetpointValues[3]
//     Term 18 (AT2050-0501)/CC Outputs/Current setpoint value Ch.5 <-> Data Pointer/CurrentSetpointValues[4]
//     Term 18 (AT2050-0501)/CC Outputs/Current setpoint value Ch.6 <-> Data Pointer/CurrentSetpointValues[5]
//     Term 18 (AT2050-0501)/CC Outputs/Current setpoint value Ch.7 <-> Data Pointer/CurrentSetpointValues[6]
//     Term 18 (AT2050-0501)/CC Outputs/Current setpoint value Ch.8 <-> Data Pointer/CurrentSetpointValues[7]
//     Term 18 (AT2050-0501)/CC Outputs/Current setpoint value Ch.9 <-> Data Pointer/CurrentSetpointValues[8]
//     Term 18 (AT2050-0501)/Term 19 (AT2050-5501)/FB Inputs/Value Channel 01 <-> Data Pointer/RawPositionValues[0]
//     Term 18 (AT2050-0501)/Term 19 (AT2050-5501)/FB Inputs/Value Channel 02 <-> Data Pointer/RawPositionValues[1]
//     Term 18 (AT2050-0501)/Term 19 (AT2050-5501)/FB Inputs/Value Channel 03 <-> Data Pointer/RawPositionValues[2]
//     Term 18 (AT2050-0501)/Term 19 (AT2050-5501)/FB Inputs/Value Channel 04 <-> Data Pointer/RawPositionValues[3]
//     Term 18 (AT2050-0501)/Term 19 (AT2050-5501)/FB Inputs/Value Channel 05 <-> Data Pointer/RawPositionValues[4]
//     Term 18 (AT2050-0501)/Term 19 (AT2050-5501)/FB Inputs/Value Channel 06 <-> Data Pointer/RawPositionValues[5]
//     Term 18 (AT2050-0501)/Term 19 (AT2050-5501)/FB Inputs/Value Channel 07 <-> Data Pointer/RawPositionValues[6]
//     Term 18 (AT2050-0501)/Term 19 (AT2050-5501)/FB Inputs/Value Channel 08 <-> Data Pointer/RawPositionValues[7]
//     Term 18 (AT2050-0501)/Term 19 (AT2050-5501)/FB Inputs/Value Channel 09 <-> Data Pointer/RawPositionValues[8]
//     Term 18 (AT2050-0501)/Term 19 (AT2050-5501)/FB Inputs/Value Channel 10 <-> Data Pointer/RawPositionValues[9]
//     Term 18 (AT2050-0501)/Term 19 (AT2050-5501)/FB Inputs/Value Channel 11 <-> Data Pointer/RawPositionValues[10]
//     Term 18 (AT2050-0501)/Term 19 (AT2050-5501)/FB Inputs/Value Channel 12 <-> Data Pointer/RawPositionValues[11]
//     Term 18 (AT2050-0501)/Term 19 (AT2050-5501)/FB Inputs/Value Channel 13 <-> Data Pointer/RawPositionValues[12]
//     Term 18 (AT2050-0501)/Term 19 (AT2050-5501)/FB Inputs/Value Channel 14 <-> Data Pointer/RawPositionValues[13]
//     Term 18 (AT2050-0501)/Term 19 (AT2050-5501)/FB Inputs/Value Channel 15 <-> Data Pointer/RawPositionValues[14]
//     Term 18 (AT2050-0501)/Term 19 (AT2050-5501)/FB Inputs/Value Channel 16 <-> Data Pointer/RawPositionValues[15]
//     Term 18 (AT2050-0501)/Term 19 (AT2050-5501)/FB Inputs/Value Channel 17 <-> Data Pointer/RawPositionValues[16]
//     Term 18 (AT2050-0501)/Term 19 (AT2050-5501)/FB Inputs/Value Channel 18 <-> Data Pointer/RawPositionValues[17]
//     Term 18 (AT2050-0501)/Term 19 (AT2050-5501)/FB Inputs/Value Channel 19 <-> Data Pointer/RawPositionValues[18]
//     Term 18 (AT2050-0501)/Term 19 (AT2050-5501)/FB Inputs/Value Channel 20 <-> Data Pointer/RawPositionValues[19]
//     Term 18 (AT2050-0501)/Term 19 (AT2050-5501)/FB Inputs/Value Channel 21 <-> Data Pointer/RawPositionValues[20]
//     Term 18 (AT2050-0501)/Term 19 (AT2050-5501)/FB Inputs/Value Channel 22 <-> Data Pointer/RawPositionValues[21]
//     Term 18 (AT2050-0501)/Term 19 (AT2050-5501)/FB Inputs/Value Channel 23 <-> Data Pointer/RawPositionValues[22]
//     Term 18 (AT2050-0501)/Term 19 (AT2050-5501)/FB Inputs/Value Channel 24 <-> Data Pointer/RawPositionValues[23]
//     Term 18 (AT2050-0501)/Term 19 (AT2050-5501)/FB Inputs/Value Channel 25 <-> Data Pointer/RawPositionValues[24]
//     Term 18 (AT2050-0501)/Term 19 (AT2050-5501)/FB Inputs/Value Channel 26 <-> Data Pointer/RawPositionValues[25]
//     Term 18 (AT2050-0501)/Term 19 (AT2050-5501)/FB Inputs/Value Channel 27 <-> Data Pointer/RawPositionValues[26]
//     Term 18 (AT2050-0501)/Term 19 (AT2050-5501)/FB Inputs/Value Channel 28 <-> Data Pointer/RawPositionValues[27]
//     Term 18 (AT2050-0501)/Term 19 (AT2050-5501)/FB Inputs/Value Channel 29 <-> Data Pointer/RawPositionValues[28]
//     Term 18 (AT2050-0501)/Term 19 (AT2050-5501)/FB Inputs/Value Channel 30 <-> Data Pointer/RawPositionValues[29]
//     Term 18 (AT2050-0501)/Term 19 (AT2050-5501)/FB Inputs/Value Channel 31 <-> Data Pointer/RawPositionValues[30]
//     Term 18 (AT2050-0501)/Term 19 (AT2050-5501)/FB Inputs/Value Channel 32 <-> Data Pointer/RawPositionValues[31]
//   (this object) <-> Device 1 (EtherCAT)/Term 1 (EK1100)/Term 3 (EL9227-5500)
//     PlcTask Inputs/MAIN.tmp <-> OCP Inputs Channel 1/Voltage In
//   (this object) <-> NC-Task 1/Axes/FeedAxis
//     PlcTask Inputs/MAIN.FeedAxis.NcToPlc <-> Outputs/ToPlc
//     PlcTask Outputs/MAIN.FeedAxis.PlcToNc <-> Inputs/FromPlc
//   (this object) <-> NC-Task 1/Axes/Mover Axis 1
//     PlcTask Inputs/MAIN.Movers[1]._Axis.NcToPlc <-> Outputs/ToPlc
//     PlcTask Outputs/MAIN.Movers[1]._Axis.PlcToNc <-> Inputs/FromPlc
//   (this object) <-> NC-Task 1/Axes/Mover Axis 2
//     PlcTask Inputs/MAIN.Movers[2]._Axis.NcToPlc <-> Outputs/ToPlc
//     PlcTask Outputs/MAIN.Movers[2]._Axis.PlcToNc <-> Inputs/FromPlc
//   (this object) <-> NC-Task 1/Axes/VirtualMaster
//     PlcTask Inputs/MAIN.VirtualMover._Axis.NcToPlc <-> Outputs/ToPlc
//     PlcTask Outputs/MAIN.VirtualMover._Axis.PlcToNc <-> Inputs/FromPlc
//   (this object) <-> NC-Task 1/Objects/Group1 (CA Group)
//     PlcTask Inputs/MAIN.Xts._AxesGroupRef.NcToPlc/CA <-> Group Outputs/ToPLC
//     PlcTask Outputs/MAIN.Xts._AxesGroupRef.PlcToNc <-> Group Inputs/FromPLC

CONFIGURATION Code
    RESOURCE PLC ON TwinCAT3
        TASK PlcTask(INTERVAL := T#2ms, PRIORITY := 20);
        PROGRAM MAIN WITH PlcTask : MAIN;
    END_RESOURCE
END_CONFIGURATION

// ---- Tests/CamBuild/ST_Camming.TcDUT
TYPE ST_Camming :
	STRUCT
		camIn		   : MC_CamIn_V2;
		camOut		   : MC_CamOut;
		camPoints	   : ARRAY[1..94] OF MC_MotionFunctionPoint;
		camRef		   : MC_CAM_REF;
		camTableSelect : MC_CamTableSelect;
		camAdd		   : MC_CamAdd;
		camRemove	   : MC_CamRemove;
        camScaling     :  ST_CamScalingData;
	END_STRUCT
END_TYPE

// ---- Tests/Base/Interface/I_SequenceTest.TcIO
INTERFACE I_SequenceTest EXTENDS I_Base, I_Cyclic

{attribute 'monitoring' := 'call'}
PROPERTY Busy : BOOL
GET
END_GET
END_PROPERTY

METHOD Reset
VAR_INPUT
END_VAR
END_METHOD

METHOD Start
VAR_INPUT
END_VAR
END_METHOD

METHOD Stop
VAR_INPUT
END_VAR
END_METHOD

END_INTERFACE

// ---- Tests/CamBuild/Interface/I_CamBuildSequence.TcIO
INTERFACE I_CamBuildSequence EXTENDS I_SequenceTest

END_INTERFACE

// ---- Tests/CamCurveCompTest/I_CamCurveComp.TcIO
INTERFACE I_CamCurveComp EXTENDS I_SequenceTest

END_INTERFACE

// ---- MAIN.TcPOU
PROGRAM MAIN
VAR
	Xts				  : XtsSystem('XTS ProcessingUnit 1');
	Movers			  : ARRAY[1..2] OF XtsMover[('Mover 1', 0, Xts), ('Mover 2', 0, Xts)];
	VirtualCollection : XtsMoverCollection;
	ReleaseTrigger	  : XtsPositionTrigger('Release Trigger', 0, VirtualCollection, Xts);
	VirtualMover	  : XtsMover('Virtual Mover', 0, Xts);
	WholeTrack		  : XtsZone('Whole Track', Xts.Movers, 0, 1500, Xts);
	MoveVelocity	  : XtsMoverMoveVelocity;
	Halt			  : XtsMoverHalt;
	tmp AT %I*		  : UINT;
	State			  : UDINT;
	Hmi				  : XtsBasicHmi<3, 1, 3, 1>('Hmi', Xts);

	//
	startVirtualPosition : LREAL;
	SetPosition			 : MC_SetPosition;
	MoveToPos			 : ARRAY[1..2] OF MC_MoveAbsolute;
	GearIn				 : ARRAY[1..2] OF MC_GearIn;
	PhaseAxis			 : ARRAY[1..2] OF MC_PhasingRelative;
	OpenCloseDistance	 : LREAL := 60;
	commandedPosition	 : ARRAY[1..2] OF LREAL;
	Gap					 : LREAL := 115;
	newPosition			 : LREAL;

	//
	PickupPosition : LREAL := 875;
	DelayTimer	   : TON;
	PrePickupTime  : TIME  := T#5S;
	PostPickupTIme : TIME  := T#2S;
	ProductSpeed   : LREAL := 400;
	OpenVelocity   : LREAL := 600;

	//Reversing Sequence
	stopReversing : BOOL;
	DwellTime	  : TIME := T#3S;
	DwellTimer	  : TON;
	Pos1		  : LREAL := 750;
	Pos2		  : LREAL := 1000;
	godotHmi	  : GodotHmi(Movers[1]);

	//BallScrew Sample
	SyncTrigger	  : XtsPositionTrigger('SyncTrigger', 750, VirtualCollection, Xts);
	DesyncTrigger : XtsPositionTrigger('DesyncTrigger', 1000, VirtualCollection, Xts);
	FeedAxis	  : AXIS_REF;
	Feeder		  : AxisPTP('Feeder', FeedAxis);
	DeSyncedSpeed : LREAL := 200;
	AxisSpeed	  : LREAL := 200;
	Mover		  : I_XtsMover;
	Pitch		  : LREAL := 50;
	SyncPosition  : LREAL := 1100;
	_NextPocket	  : UDINT;

	// Cam Generator
	CurveComp	   : CamBuild;
	MoverCurveComp : CamCurveComp;
	MultiCamComp   : SplitCamBuild;
	MultiCamTest   : SplitCamRun;
END_VAR

IF NOT Xts.Initialized OR NOT Feeder.Initialized THEN
	Feeder.Initialize();
	Xts.Initialize();
	Xts.Parameters.Velocity		 := 200;
	Xts.Parameters.Acceleration	 := 5_000;
	Xts.Parameters.Deceleration	 := 5_000;
	Xts.Parameters.Jerk			 := 100_000;
	Xts.Parameters.Gap			 := 100;
	VirtualMover.VirtualMover	 := TRUE;
	Movers[1].ManualGroupControl := TRUE;
	Movers[2].ManualGroupControl := TRUE;
	Hmi.BuildHMI();
	IF VirtualCollection.IsEmpty THEN
		VirtualCollection.AddItem(VirtualMover);
	END_IF

	RETURN;
END_IF

CASE State OF
	0:
	1:
		Xts.Reset();
		Xts.ResetMovers();
		State := 0;

	5:
		Xts.Utility.SetConfiguredDetectionCount(Xts.Utility.GetDetectedMoverCount());
		State := 1;

	10:
		Xts.Enable();
		IF Xts.Enabled THEN
			State := 50;
		END_IF

	20:
		Xts.Disable();
		IF NOT Xts.Enabled THEN
			State := 0;
		END_IF

	60:
		MoveVelocity.CopyParametersFrom(Xts.Parameters);
		MoveVelocity.ExecuteOn(Xts);
		State := 50;

	61:
		Halt.CopyParametersFrom(Xts.Parameters);
		Halt.ExecuteOn(Xts);
		State := 50;

	70:
		MoveVelocity.CopyParametersFrom(Xts.Parameters);
		MoveVelocity.ExecuteOn(VirtualMover);
		State := 50;

	71:
		Halt.CopyParametersFrom(Xts.Parameters);
		Halt.ExecuteOn(VirtualMover);
		State := 50;

	100:
		IF Xts.Utility.GetMoverIdDetectionState() <> MoverIdDetectionStateEnum.Valid THEN
			State := 101;
		ELSE
			State := 111;
		END_IF

	101:
		Xts.Enable();
		IF Xts.Enabled THEN
			State := 102;
		END_IF

	102:
		Xts.Disable();
		IF NOT Xts.Enabled THEN
			State := 100;
		END_IF

	110:
		Xts.Disable();
		IF NOT Xts.Enabled THEN
			State := 111;
		END_IF

	111:
		//startVirtualPosition := (Movers[2].Position - Movers[1].Position) / 2 + Movers[1].Position;
		startVirtualPosition := 59;
		SetPosition(Axis := VirtualMover.Axis, Position := startVirtualPosition, Execute := TRUE);
		IF SetPosition.Done OR SetPosition.Error THEN
			State := 120;
			SetPosition(Axis := VirtualMover.Axis, Execute := FALSE);
		END_IF

	120:
		Xts.Enable();
		IF Xts.Enabled THEN
			State := 122;
		END_IF

	121:
		VirtualMover.Parameters.CopyFrom(Xts.Parameters);
		VirtualMover.Parameters.Gap := 0;
		VirtualMover.MoveToPosition(VirtualMover.Position);
		Movers[1].Parameters.CopyFrom(Xts.Parameters);
		Movers[2].Parameters.CopyFrom(Xts.Parameters);
		commandedPosition[1] := startVirtualPosition - Gap;
		commandedPosition[2] := startVirtualPosition + Gap;
		MoveToPos[1](Axis		  := Movers[1].Axis,
					 Execute	  := TRUE,
					 Position	  := commandedPosition[1],
					 Velocity	  := 300,
					 Acceleration := 5000,
					 Deceleration := 5000,
					 Jerk		  := 100000);

		MoveToPos[2](Axis		  := Movers[2].Axis,
					 Execute	  := TRUE,
					 Position	  := commandedPosition[2],
					 Velocity	  := 300,
					 Acceleration := 5000,
					 Deceleration := 5000,
					 Jerk		  := 100000);

		IF MoveToPos[1].Error OR MoveToPos[2].Error OR (MoveToPos[1].Done AND MoveToPos[2].Done) THEN
			MoveToPos[1](Axis := Movers[1].Axis, Execute := FALSE);
			MoveToPos[2](Axis := Movers[2].Axis, Execute := FALSE);
			State := 125;
		END_IF

	122:
		VirtualMover.Parameters.CopyFrom(Xts.Parameters);
		VirtualMover.Parameters.Gap := 0;
		VirtualMover.MoveToPosition(VirtualMover.Position);
		Movers[1].Parameters.CopyFrom(Xts.Parameters);
		Movers[2].Parameters.CopyFrom(Xts.Parameters);
		commandedPosition[1] := 115;
		commandedPosition[2] := commandedPosition[1] - Gap;
		MoveToPos[1](Axis		  := Movers[1].Axis,
					 Execute	  := TRUE,
					 Position	  := commandedPosition[1] + TRUNC(Movers[1].Axis.NcToPlc.ActPos / 1500.0) * 1500,
					 Velocity	  := 300,
					 Acceleration := 5000,
					 Deceleration := 5000,
					 Jerk		  := 100000);

		MoveToPos[2](Axis		  := Movers[2].Axis,
					 Execute	  := TRUE,
					 Position	  := commandedPosition[2] + TRUNC(Movers[1].Axis.NcToPlc.ActPos / 1500.0) * 1500,
					 Velocity	  := 300,
					 Acceleration := 5000,
					 Deceleration := 5000,
					 Jerk		  := 100000);

		IF MoveToPos[1].Error OR MoveToPos[2].Error OR (MoveToPos[1].Done AND MoveToPos[2].Done) THEN
			MoveToPos[1](Axis := Movers[1].Axis, Execute := FALSE);
			MoveToPos[2](Axis := Movers[2].Axis, Execute := FALSE);
			State := 125;
		END_IF

	125:
		GearIn[1](Master	   := VirtualMover.Axis,
				  Slave		   := Movers[1].Axis,
				  Execute	   := TRUE,
				  Acceleration := 10_000,
				  Deceleration := 10_000,
				  Jerk		   := 100_000);

		GearIn[2](Master	   := VirtualMover.Axis,
				  Slave		   := Movers[2].Axis,
				  Execute	   := FALSE,
				  Acceleration := 10_000,
				  Deceleration := 10_000,
				  Jerk		   := 100_000);

		IF GearIn[1].InGear (*AND GearIn[2].InGear *) THEN
			GearIn[1](Master := VirtualMover.Axis, Slave := Movers[1].Axis, Execute := FALSE);
			GearIn[2](Master := VirtualMover.Axis, Slave := Movers[2].Axis, Execute := FALSE);
			State := 150;
		END_IF

	130:
		VirtualMover.Parameters.CopyFrom(Xts.Parameters);
		VirtualMover.MoveToPosition(newPosition, XtsCore.Tc3_Mc3Definitions.MC_DIRECTION.mcDirectionShortestWay);
		State := 150;

	135:
		VirtualMover.Parameters.CopyFrom(Xts.Parameters);
		VirtualMover.MoveVelocity(Xts.Parameters.Velocity);
		State := 150;

	136:
		VirtualMover.Halt(Xts.Parameters.Deceleration, Xts.Parameters.Gap);
		State := 150;

	//Reversing Sequence 150-155
	160:
		VirtualMover.Parameters.CopyFrom(Xts.Parameters);
		VirtualMover.MoveToPosition(Pos1, XtsCore.Tc3_Mc3Definitions.MC_DIRECTION.mcDirectionShortestWay);
		State := 161;

	161:
		DwellTimer(IN := VirtualMover.InPosition, PT := DwellTime);
		IF DwellTimer.Q THEN
			DwellTimer(IN := FALSE);
			State := 162;
		END_IF

	162:
		VirtualMover.Parameters.CopyFrom(Xts.Parameters);
		VirtualMover.MoveToPosition(Pos2, XtsCore.Tc3_Mc3Definitions.MC_DIRECTION.mcDirectionShortestWay);
		State := 163;

	163:
		DwellTimer(IN := VirtualMover.InPosition, PT := DwellTime);
		IF DwellTimer.Q THEN
			DwellTimer(IN := FALSE);
			State := 164;
		END_IF

	164:
		IF stopReversing THEN
			stopReversing := FALSE;
			State		  := 150;
		ELSE
			State := 160;
		END_IF

	140:
		PhaseAxis[1](Master		  := VirtualMover.Axis,
					 Slave		  := Movers[1].Axis,
					 Execute	  := TRUE,
					 PhaseShift	  := OpenCloseDistance,
					 Velocity	  := Xts.Parameters.Velocity * 1.2,
					 Acceleration := 10_000,
					 Deceleration := 10_000,
					 Jerk		  := 100_000);

		PhaseAxis[2](Master		  := VirtualMover.Axis,
					 Slave		  := Movers[2].Axis,
					 Execute	  := FALSE,
					 PhaseShift	  := OpenCloseDistance,
					 Velocity	  := Xts.Parameters.Velocity * 1.2,
					 Acceleration := 10_000,
					 Deceleration := 10_000,
					 Jerk		  := 100_000);

		IF PhaseAxis[1].Error OR PhaseAxis[1].Done THEN
			PhaseAxis[1](Master := VirtualMover.Axis, Slave := Movers[1].Axis, Execute := FALSE);
			PhaseAxis[2](Master := VirtualMover.Axis, Slave := Movers[2].Axis, Execute := FALSE);
			State := 150;
		END_IF

	200:
		//Move to pick up position

		//Wait at pickup up position for PickupTime

		//Phase to close and pickup the ball

		//Move velocity

		//Trigger Active, tell Mover[1] to phase open distance
		//Phase Done, go back to repeat
		VirtualMover.MoveToPosition(PickupPosition);
		IF NOT VirtualMover.CurrentTask.Busy AND VirtualMover.InPosition THEN
			State := 210;
		END_IF

	210:
		DelayTimer(IN := TRUE, PT := PrePickupTime);
		IF DelayTimer.Q THEN
			DelayTimer(IN := FALSE);
			State := 211;
		END_IF

	211:
		PhaseAxis[1](Master		  := VirtualMover.Axis,
					 Slave		  := Movers[1].Axis,
					 Execute	  := TRUE,
					 PhaseShift	  := OpenCloseDistance,
					 Velocity	  := Xts.Parameters.Velocity * 1.2,
					 Acceleration := 10_000,
					 Deceleration := 10_000,
					 Jerk		  := 100_000);

		IF PhaseAxis[1].Error OR PhaseAxis[1].Done THEN
			PhaseAxis[1](Master := VirtualMover.Axis, Slave := Movers[1].Axis, Execute := FALSE);
			State := 212;
		END_IF

	212:
		DelayTimer(IN := TRUE, PT := PostPickupTime);
		IF DelayTimer.Q THEN
			DelayTimer(IN := FALSE);
			VirtualMover.MoveVelocity(ProductSpeed);
			State := 213;
		END_IF

	213:
		IF ReleaseTrigger.MoverIsPresent THEN
			ReleaseTrigger.GetMover();
			State := 220;
		END_IF

	220:
		PhaseAxis[1](Master		  := VirtualMover.Axis,
					 Slave		  := Movers[1].Axis,
					 Execute	  := TRUE,
					 PhaseShift	  := -OpenCloseDistance,
					 Velocity	  := OpenVelocity,
					 Acceleration := 10_000,
					 Deceleration := 10_000,
					 Jerk		  := 100_000);

		IF PhaseAxis[1].Error OR PhaseAxis[1].Done THEN
			PhaseAxis[1](Master := VirtualMover.Axis, Slave := Movers[1].Axis, Execute := FALSE);
			State := 200;
		END_IF

	//Start of the BallScrew Sample Code
	300:
		//Set Master Position to 0
		Feeder.Home();
		IF NOT Feeder.Busy THEN
			State := 301;
		END_IF

	301:
		//Enable Master
		Feeder.Enable();
		IF Feeder.Enabled THEN
			State := 302;
		END_IF

	302:
		//enable the PosTrigger
		SyncTrigger.Enable();
		IF SyncTrigger.Enabled THEN
			State := 303;
			SyncTrigger.MoverQueue.Clear();
		END_IF

	303:
		//MoveVelocity on Master
		VirtualMover.MoveVelocity(DeSyncedSpeed);
		Feeder.MoveVelocity(AxisSpeed);
		State := 305;

	305:
		_NextPocket := DINT_TO_UDINT(TRUNC(Feeder.SetPosition / Pitch) + 1);
		//Monitor Trigger
		IF SyncTrigger.MoverIsPresent THEN
			Mover														  := SyncTrigger.GetMover();
			Mover.Parameters.Velocity									  := AxisSpeed * 2;
			Mover.Parameters.Acceleration								  := 10_000;
			Mover.Parameters.Deceleration								  := 10_000;
			Mover.Parameters.Jerk										  := 100_000;
			Mover.Parameters.SyncAxis.Options_CA.DirectionReversalAllowed := FALSE;
			Mover.Parameters.SyncAxis.SyncMode							  := XtsCore.Tc3_McCollisionAvoidance.MC_SYNC_MODE.mcSyncModePositive;
			Mover.SyncToAxis(Master := FeedAxis, MasterSyncPosition := _NextPocket * Pitch, SlaveSyncPosition := SyncPosition); //TOOD: Fix Position calcs
		END_IF

		IF DeSyncTrigger.MoverIsPresent THEN
			Mover := DeSyncTrigger.GetMover();
			Mover.MoveVelocity(DeSyncedSpeed);
		END_IF

	310:
		//Disable Trigger
		SyncTrigger.Disable();

		//Stop Master
		Feeder.Stop();
		IF Feeder.Stopped THEN
			State := 311;
		END_IF

	311:
		//Stop Zone
		VirtualMover.Halt(Xts.Parameters.Deceleration, Xts.Parameters.Gap);
		State := 312;

	312:
		IF NOT Halt.Busy THEN
			State := 313;
		END_IF

	313:
		Feeder.Disable();
		//Disable Master		
		IF NOT Feeder.Enabled THEN
			State := 150;
		END_IF

	401:
		CurveComp.Start();
		SetStep(State, 400);

	402:
		CurveComp.Reset();
		SetStep(State, 400);

	403:
		MultiCamComp.Start();
		SetStep(State, 400);

	404:
		MultiCamComp.Reset();
		SetStep(State, 400);

	410:
		MoverCurveComp.FrontMover	:= Movers[1];
		MoverCurveComp.RearMover	:= Movers[2];
		MoverCurveComp.VirtualMover := VirtualMover;
		MoverCurveComp.Start();
		NextMinorStep(State);

	411:
		IF NOT MoverCurveComp.Busy THEN
			SetStep(State, 400);
		END_IF

	412:
		MoverCurveComp.Reset();
		SetStep(State, 400);

	420:
		MultiCamTest.FrontMover	  := Movers[1];
		MultiCamTest.RearMover	  := Movers[2];
		MultiCamTest.VirtualMover := VirtualMover;
		MultiCamTest.Start();
		NextMinorStep(State);

	421:
		IF NOT MultiCamTest.Busy THEN
			SetStep(State, 400);
		END_IF

	422:
		MultiCamTest.Reset();
		SetStep(State, 400);
END_CASE

MultiCamComp.CyclicLogic();
MultiCamTest.CyclicLogic();
MoverCurveComp.CyclicLogic();
CurveComp.CyclicLogic();
Feeder.CyclicLogic();
godotHmi.CyclicLogic();
Xts.CyclicLogic();
Hmi.CyclicLogic();

END_PROGRAM

// ---- POUs/GodotHmi.TcPOU
FUNCTION_BLOCK GodotHmi
VAR
	_Mover : I_XtsMover;
	{attribute 'godot'}
	productPosition : LREAL;
	{attribute 'godot'}
	setVelocity	  : LREAL;
	tccomPosition : LREAL;
END_VAR

METHOD CyclicLogic
VAR_INPUT
END_VAR
VAR_INST
	PositionInfo : REFERENCE TO XtsCore.Tc3_XTS_Utility.ST_PositionInfo;
END_VAR
productPosition := _Mover.Position;
setVelocity		:= _Mover.Axis.NcToPlc.SetVelo;
PositionInfo	REF= _Mover.MoverUtility.GetPositionInfo();
tccomPosition	:= PositionInfo.fTrackPosition;
END_METHOD

//FB_Init is always available implicitly and it is used primarily for initialization.

//The return value is not evaluated. For a specific influence, you can also declare the

//methods explicitly and provide additional code there with the standard initialization

//code. You can evaluate the return value.
METHOD FB_Init : BOOL
VAR_INPUT
	bInitRetains : BOOL; // TRUE: the retain variables are initialized (reset warm / reset cold)
	bInCopyCode	 : BOOL; // TRUE: the instance will be copied to the copy code afterward (online change)   
	Mover		 : I_XtsMover;
END_VAR
_Mover := Mover;
END_METHOD

END_FUNCTION_BLOCK

// ---- Godot.TcPOU
PROGRAM Godot
VAR
	on : BOOL;
	//_Godot : GodotHmi(Main.Movers[1]);
END_VAR

IF NOT on THEN
	RETURN;
END_IF

//_Godot.CyclicLogic();

END_PROGRAM

// ---- Tests/CamBuild/CamBuild.TcPOU
FUNCTION_BLOCK CamBuild IMPLEMENTS I_CamBuildSequence
VAR
	_State	 : UDINT;
	_Camming : ST_Camming;
	point	 : UDINT;
	_Custom	 : BOOL;
END_VAR

{attribute 'monitoring' := 'call'}
PROPERTY Busy : BOOL
GET
Busy := _State <> 0;
END_GET
END_PROPERTY

METHOD CyclicLogic
VAR_INPUT
END_VAR
CASE _State OF
	0:
	10:
		IF NOT _Custom THEN
			// Clothoid oval cam, 9 points, generated from cam-table.json.

			// Master = position along the orange (outer, 99 mm offset) path.

			// Slave  = position along the blue (track centreline) path.

			// Periodic: 1061.0177 mm of master -> 750.0000 mm of slave,

			// which is half a lap. Run it twice for a full lap.

			// Worst deviation from the exact clothoid: 2.3 um.

			// Master zero is where the left curve meets the bottom straight.
			// Carrier A enters at master 65 mm, carrier B at 180 mm.
			point												  := 1;
			_Camming.camPoints[point].MasterPos		  := 0.0000;
			_Camming.camPoints[point].SlavePos		  := 0.0000;
			_Camming.camPoints[point].PointIndex		  := point;
			_Camming.camPoints[point].FunctionType	  := MC_MotionFunctionType.MOTIONFUNCTYPE_POLYNOM1;
			_Camming.camPoints[point].PointType		  := MC_MotionPointType.MOTIONPOINTTYPE_ACTIVATION;
			_Camming.camPoints[point].RelIndexNextPoint := 1;
			_Camming.camPoints[point].SlaveVelo		  := 1.0000000;
			_Camming.camPoints[point].SlaveAcc		  := 0.004928218;
			_Camming.camPoints[point].SlaveJerk		  := 0.00;
			point												  := 2;
			_Camming.camPoints[point].MasterPos		  := 250.0000;
			_Camming.camPoints[point].SlavePos		  := 250.0000;
			_Camming.camPoints[point].PointIndex		  := point;
			_Camming.camPoints[point].FunctionType	  := MC_MotionFunctionType.MOTIONFUNCTYPE_POLYNOM5_MM;
			_Camming.camPoints[point].PointType		  := MC_MotionPointType.MOTIONPOINTTYPE_MOTION;
			_Camming.camPoints[point].RelIndexNextPoint := 1;
			_Camming.camPoints[point].SlaveVelo		  := 1.0000000;
			_Camming.camPoints[point].SlaveAcc		  := -0.004928218;
			_Camming.camPoints[point].SlaveJerk		  := 0.00;
			point												  := 3;
			_Camming.camPoints[point].MasterPos		  := 362.2284;
			_Camming.camPoints[point].SlavePos		  := 341.4293;
			_Camming.camPoints[point].PointIndex		  := point;
			_Camming.camPoints[point].FunctionType	  := MC_MotionFunctionType.MOTIONFUNCTYPE_POLYNOM5_MM;
			_Camming.camPoints[point].PointType		  := MC_MotionPointType.MOTIONPOINTTYPE_MOTION;
			_Camming.camPoints[point].RelIndexNextPoint := 1;
			_Camming.camPoints[point].SlaveVelo		  := 0.6872957;
			_Camming.camPoints[point].SlaveAcc		  := -0.001602554;
			_Camming.camPoints[point].SlaveJerk		  := 0.00;
			point												  := 4;
			_Camming.camPoints[point].MasterPos		  := 603.2346;
			_Camming.camPoints[point].SlavePos		  := 476.0707;
			_Camming.camPoints[point].PointIndex		  := point;
			_Camming.camPoints[point].FunctionType	  := MC_MotionFunctionType.MOTIONFUNCTYPE_POLYNOM5_MM;
			_Camming.camPoints[point].PointType		  := MC_MotionPointType.MOTIONPOINTTYPE_MOTION;
			_Camming.camPoints[point].RelIndexNextPoint := 1;
			_Camming.camPoints[point].SlaveVelo		  := 0.4705900;
			_Camming.camPoints[point].SlaveAcc		  := -0.000509905;
			_Camming.camPoints[point].SlaveJerk		  := 0.00;
			point												  := 5;
			_Camming.camPoints[point].MasterPos		  := 637.0257;
			_Camming.camPoints[point].SlavePos		  := 491.6870;
			_Camming.camPoints[point].PointIndex		  := point;
			_Camming.camPoints[point].FunctionType	  := MC_MotionFunctionType.MOTIONFUNCTYPE_POLYNOM5_MM;
			_Camming.camPoints[point].PointType		  := MC_MotionPointType.MOTIONPOINTTYPE_MOTION;
			_Camming.camPoints[point].RelIndexNextPoint := 1;
			_Camming.camPoints[point].SlaveVelo		  := 0.4539877;
			_Camming.camPoints[point].SlaveAcc		  := -0.000357875;
			_Camming.camPoints[point].SlaveJerk		  := 0.00;
			point												  := 6;
			_Camming.camPoints[point].MasterPos		  := 673.9920;
			_Camming.camPoints[point].SlavePos		  := 508.3130;
			_Camming.camPoints[point].PointIndex		  := point;
			_Camming.camPoints[point].FunctionType	  := MC_MotionFunctionType.MOTIONFUNCTYPE_POLYNOM5_MM;
			_Camming.camPoints[point].PointType		  := MC_MotionPointType.MOTIONPOINTTYPE_MOTION;
			_Camming.camPoints[point].RelIndexNextPoint := 1;
			_Camming.camPoints[point].SlaveVelo		  := 0.4539877;
			_Camming.camPoints[point].SlaveAcc		  := 0.000357875;
			_Camming.camPoints[point].SlaveJerk		  := 0.00;
			point												  := 7;
			_Camming.camPoints[point].MasterPos		  := 707.7831;
			_Camming.camPoints[point].SlavePos		  := 523.9293;
			_Camming.camPoints[point].PointIndex		  := point;
			_Camming.camPoints[point].FunctionType	  := MC_MotionFunctionType.MOTIONFUNCTYPE_POLYNOM5_MM;
			_Camming.camPoints[point].PointType		  := MC_MotionPointType.MOTIONPOINTTYPE_MOTION;
			_Camming.camPoints[point].RelIndexNextPoint := 1;
			_Camming.camPoints[point].SlaveVelo		  := 0.4705900;
			_Camming.camPoints[point].SlaveAcc		  := 0.000509905;
			_Camming.camPoints[point].SlaveJerk		  := 0.00;
			point												  := 8;
			_Camming.camPoints[point].MasterPos		  := 948.7893;
			_Camming.camPoints[point].SlavePos		  := 658.5707;
			_Camming.camPoints[point].PointIndex		  := point;
			_Camming.camPoints[point].FunctionType	  := MC_MotionFunctionType.MOTIONFUNCTYPE_POLYNOM5_MM;
			_Camming.camPoints[point].PointType		  := MC_MotionPointType.MOTIONPOINTTYPE_MOTION;
			_Camming.camPoints[point].RelIndexNextPoint := 1;
			_Camming.camPoints[point].SlaveVelo		  := 0.6872957;
			_Camming.camPoints[point].SlaveAcc		  := 0.001602554;
			_Camming.camPoints[point].SlaveJerk		  := 0.00;
			point												  := 9;
			_Camming.camPoints[point].MasterPos		  := 1061.0177;
			_Camming.camPoints[point].SlavePos		  := 750.0000;
			_Camming.camPoints[point].PointIndex		  := point;
			_Camming.camPoints[point].FunctionType	  := MC_MotionFunctionType.MOTIONFUNCTYPE_POLYNOM1;
			_Camming.camPoints[point].PointType		  := MC_MotionPointType.MOTIONPOINTTYPE_MOTION;
			_Camming.camPoints[point].RelIndexNextPoint := 0;
			_Camming.camPoints[point].SlaveVelo		  := 1.0000000;
			_Camming.camPoints[point].SlaveAcc		  := 0.004928218;
			_Camming.camPoints[point].SlaveJerk		  := 0.00;
			_Camming.camRef.NoOfColumns				  := 1;
			_Camming.camRef.NoOfRows					  := point;
			_Camming.camRef.TableType					  := MC_TableType.MC_TABLETYPE_MOTIONFUNCTION;
			_Camming.camRef.ArraySize					  := SIZEOF(_Camming.camPoints);
			_Camming.camRef.pArray					  := ADR(_Camming.camPoints);
            
        END_IF
		//
		_Camming.camRef.NoOfColumns := 1;
		_Camming.camRef.NoOfRows	:= point;
		_Camming.camRef.TableType	:= MC_TableType.MC_TABLETYPE_MOTIONFUNCTION;
		_Camming.camRef.ArraySize	:= SIZEOF(_Camming.camPoints);
		_Camming.camRef.pArray		:= ADR(_Camming.camPoints);

		//
		_Camming.camTableSelect(CamTable   := _Camming.camRef,
								Execute	   := TRUE,
								Periodic   := TRUE,
								CamTableID := 1);

		IF _Camming.camTableSelect.Done THEN
			Trace.Info(__POUNAME(), 'Curve Cam Built - ID 1');
			_Camming.camTableSelect(CamTable := _Camming.camRef, Execute := FALSE);
			SetStep(_State, 0);
		END_IF
END_CASE
END_METHOD

METHOD MultiplePoints
VAR_INPUT
END_VAR
point										:= 1;
_Camming.camPoints[point].MasterPos			:= 180.000;
_Camming.camPoints[point].SlavePos			:= 65.000;
_Camming.camPoints[point].PointIndex		:= point;
_Camming.camPoints[point].FunctionType		:= MC_MotionFunctionType.MOTIONFUNCTYPE_POLYNOM5_MM;
_Camming.camPoints[point].PointType			:= MC_MotionPointType.MOTIONPOINTTYPE_ACTIVATION;
_Camming.camPoints[point].RelIndexNextPoint := 1;
_Camming.camPoints[point].SlaveVelo			:= 1.000000;
_Camming.camPoints[point].SlaveAcc			:= 0.00000000;
_Camming.camPoints[point].SlaveJerk			:= 0.00;

//
point										:= 2;
_Camming.camPoints[point].MasterPos			:= 250.500;
_Camming.camPoints[point].SlavePos			:= 135.500;
_Camming.camPoints[point].PointIndex		:= point;
_Camming.camPoints[point].FunctionType		:= MC_MotionFunctionType.MOTIONFUNCTYPE_POLYNOM5_MM;
_Camming.camPoints[point].PointType			:= MC_MotionPointType.MOTIONPOINTTYPE_MOTION;
_Camming.camPoints[point].RelIndexNextPoint := 1;
_Camming.camPoints[point].SlaveVelo			:= 1.000000;
_Camming.camPoints[point].SlaveAcc			:= 0.00000000;
_Camming.camPoints[point].SlaveJerk			:= 0.00;

//
point										:= 3;
_Camming.camPoints[point].MasterPos			:= 260.367;
_Camming.camPoints[point].SlavePos			:= 145.398;
_Camming.camPoints[point].PointIndex		:= point;
_Camming.camPoints[point].FunctionType		:= MC_MotionFunctionType.MOTIONFUNCTYPE_POLYNOM5_MM;
_Camming.camPoints[point].PointType			:= MC_MotionPointType.MOTIONPOINTTYPE_MOTION;
_Camming.camPoints[point].RelIndexNextPoint := 1;
_Camming.camPoints[point].SlaveVelo			:= 1.011583;
_Camming.camPoints[point].SlaveAcc			:= 0.00312668;
_Camming.camPoints[point].SlaveJerk			:= 0.00;

//
point										:= 4;
_Camming.camPoints[point].MasterPos			:= 270.233;
_Camming.camPoints[point].SlavePos			:= 155.622;
_Camming.camPoints[point].PointIndex		:= point;
_Camming.camPoints[point].FunctionType		:= MC_MotionFunctionType.MOTIONFUNCTYPE_POLYNOM5_MM;
_Camming.camPoints[point].PointType			:= MC_MotionPointType.MOTIONPOINTTYPE_MOTION;
_Camming.camPoints[point].RelIndexNextPoint := 1;
_Camming.camPoints[point].SlaveVelo			:= 1.070556;
_Camming.camPoints[point].SlaveAcc			:= 0.00898229;
_Camming.camPoints[point].SlaveJerk			:= 0.00;

//
point										:= 5;
_Camming.camPoints[point].MasterPos			:= 280.100;
_Camming.camPoints[point].SlavePos			:= 166.716;
_Camming.camPoints[point].PointIndex		:= point;
_Camming.camPoints[point].FunctionType		:= MC_MotionFunctionType.MOTIONFUNCTYPE_POLYNOM5_MM;
_Camming.camPoints[point].PointType			:= MC_MotionPointType.MOTIONPOINTTYPE_MOTION;
_Camming.camPoints[point].RelIndexNextPoint := 1;
_Camming.camPoints[point].SlaveVelo			:= 1.187356;
_Camming.camPoints[point].SlaveAcc			:= 0.01442322;
_Camming.camPoints[point].SlaveJerk			:= 0.00;

//
point										:= 6;
_Camming.camPoints[point].MasterPos			:= 289.967;
_Camming.camPoints[point].SlavePos			:= 179.194;
_Camming.camPoints[point].PointIndex		:= point;
_Camming.camPoints[point].FunctionType		:= MC_MotionFunctionType.MOTIONFUNCTYPE_POLYNOM5_MM;
_Camming.camPoints[point].PointType			:= MC_MotionPointType.MOTIONPOINTTYPE_MOTION;
_Camming.camPoints[point].RelIndexNextPoint := 1;
_Camming.camPoints[point].SlaveVelo			:= 1.346759;
_Camming.camPoints[point].SlaveAcc			:= 0.01732695;
_Camming.camPoints[point].SlaveJerk			:= 0.00;

//
point										:= 7;
_Camming.camPoints[point].MasterPos			:= 299.833;
_Camming.camPoints[point].SlavePos			:= 193.327;
_Camming.camPoints[point].PointIndex		:= point;
_Camming.camPoints[point].FunctionType		:= MC_MotionFunctionType.MOTIONFUNCTYPE_POLYNOM5_MM;
_Camming.camPoints[point].PointType			:= MC_MotionPointType.MOTIONPOINTTYPE_MOTION;
_Camming.camPoints[point].RelIndexNextPoint := 1;
_Camming.camPoints[point].SlaveVelo			:= 1.516335;
_Camming.camPoints[point].SlaveAcc			:= 0.01633779;
_Camming.camPoints[point].SlaveJerk			:= 0.00;

//
point										:= 8;
_Camming.camPoints[point].MasterPos			:= 309.700;
_Camming.camPoints[point].SlavePos			:= 209.017;
_Camming.camPoints[point].PointIndex		:= point;
_Camming.camPoints[point].FunctionType		:= MC_MotionFunctionType.MOTIONFUNCTYPE_POLYNOM5_MM;
_Camming.camPoints[point].PointType			:= MC_MotionPointType.MOTIONPOINTTYPE_MOTION;
_Camming.camPoints[point].RelIndexNextPoint := 1;
_Camming.camPoints[point].SlaveVelo			:= 1.655944;
_Camming.camPoints[point].SlaveAcc			:= 0.01140889;
_Camming.camPoints[point].SlaveJerk			:= 0.00;

//
point										:= 9;
_Camming.camPoints[point].MasterPos			:= 319.567;
_Camming.camPoints[point].SlavePos			:= 225.802;
_Camming.camPoints[point].PointIndex		:= point;
_Camming.camPoints[point].FunctionType		:= MC_MotionFunctionType.MOTIONFUNCTYPE_POLYNOM5_MM;
_Camming.camPoints[point].PointType			:= MC_MotionPointType.MOTIONPOINTTYPE_MOTION;
_Camming.camPoints[point].RelIndexNextPoint := 1;
_Camming.camPoints[point].SlaveVelo			:= 1.735262;
_Camming.camPoints[point].SlaveAcc			:= 0.00466021;
_Camming.camPoints[point].SlaveJerk			:= 0.00;

//
point										:= 10;
_Camming.camPoints[point].MasterPos			:= 329.433;
_Camming.camPoints[point].SlavePos			:= 243.059;
_Camming.camPoints[point].PointIndex		:= point;
_Camming.camPoints[point].FunctionType		:= MC_MotionFunctionType.MOTIONFUNCTYPE_POLYNOM5_MM;
_Camming.camPoints[point].PointType			:= MC_MotionPointType.MOTIONPOINTTYPE_MOTION;
_Camming.camPoints[point].RelIndexNextPoint := 1;
_Camming.camPoints[point].SlaveVelo			:= 1.755026;
_Camming.camPoints[point].SlaveAcc			:= 0.00009489;
_Camming.camPoints[point].SlaveJerk			:= 0.00;

//
point										:= 11;
_Camming.camPoints[point].MasterPos			:= 339.300;
_Camming.camPoints[point].SlavePos			:= 260.346;
_Camming.camPoints[point].PointIndex		:= point;
_Camming.camPoints[point].FunctionType		:= MC_MotionFunctionType.MOTIONFUNCTYPE_POLYNOM5_MM;
_Camming.camPoints[point].PointType			:= MC_MotionPointType.MOTIONPOINTTYPE_MOTION;
_Camming.camPoints[point].RelIndexNextPoint := 1;
_Camming.camPoints[point].SlaveVelo			:= 1.737154;
_Camming.camPoints[point].SlaveAcc			:= -0.00845956;
_Camming.camPoints[point].SlaveJerk			:= 0.00;

//
point										:= 12;
_Camming.camPoints[point].MasterPos			:= 349.167;
_Camming.camPoints[point].SlavePos			:= 276.699;
_Camming.camPoints[point].PointIndex		:= point;
_Camming.camPoints[point].FunctionType		:= MC_MotionFunctionType.MOTIONFUNCTYPE_POLYNOM5_MM;
_Camming.camPoints[point].PointType			:= MC_MotionPointType.MOTIONPOINTTYPE_MOTION;
_Camming.camPoints[point].RelIndexNextPoint := 1;
_Camming.camPoints[point].SlaveVelo			:= 1.547397;
_Camming.camPoints[point].SlaveAcc			:= -0.02615257;
_Camming.camPoints[point].SlaveJerk			:= 0.00;

//
point										:= 13;
_Camming.camPoints[point].MasterPos			:= 359.033;
_Camming.camPoints[point].SlavePos			:= 290.717;
_Camming.camPoints[point].PointIndex		:= point;
_Camming.camPoints[point].FunctionType		:= MC_MotionFunctionType.MOTIONFUNCTYPE_POLYNOM5_MM;
_Camming.camPoints[point].PointType			:= MC_MotionPointType.MOTIONPOINTTYPE_MOTION;
_Camming.camPoints[point].RelIndexNextPoint := 1;
_Camming.camPoints[point].SlaveVelo			:= 1.302751;
_Camming.camPoints[point].SlaveAcc			:= -0.02131854;
_Camming.camPoints[point].SlaveJerk			:= 0.00;

//
point										:= 14;
_Camming.camPoints[point].MasterPos			:= 368.900;
_Camming.camPoints[point].SlavePos			:= 302.681;
_Camming.camPoints[point].PointIndex		:= point;
_Camming.camPoints[point].FunctionType		:= MC_MotionFunctionType.MOTIONFUNCTYPE_POLYNOM5_MM;
_Camming.camPoints[point].PointType			:= MC_MotionPointType.MOTIONPOINTTYPE_MOTION;
_Camming.camPoints[point].RelIndexNextPoint := 1;
_Camming.camPoints[point].SlaveVelo			:= 1.136789;
_Camming.camPoints[point].SlaveAcc			:= -0.01261846;
_Camming.camPoints[point].SlaveJerk			:= 0.00;

//
point										:= 15;
_Camming.camPoints[point].MasterPos			:= 378.767;
_Camming.camPoints[point].SlavePos			:= 313.397;
_Camming.camPoints[point].PointIndex		:= point;
_Camming.camPoints[point].FunctionType		:= MC_MotionFunctionType.MOTIONFUNCTYPE_POLYNOM5_MM;
_Camming.camPoints[point].PointType			:= MC_MotionPointType.MOTIONPOINTTYPE_MOTION;
_Camming.camPoints[point].RelIndexNextPoint := 1;
_Camming.camPoints[point].SlaveVelo			:= 1.045962;
_Camming.camPoints[point].SlaveAcc			:= -0.00622413;
_Camming.camPoints[point].SlaveJerk			:= 0.00;

//
point										:= 16;
_Camming.camPoints[point].MasterPos			:= 388.633;
_Camming.camPoints[point].SlavePos			:= 323.492;
_Camming.camPoints[point].PointIndex		:= point;
_Camming.camPoints[point].FunctionType		:= MC_MotionFunctionType.MOTIONFUNCTYPE_POLYNOM5_MM;
_Camming.camPoints[point].PointType			:= MC_MotionPointType.MOTIONPOINTTYPE_MOTION;
_Camming.camPoints[point].RelIndexNextPoint := 1;
_Camming.camPoints[point].SlaveVelo			:= 1.007263;
_Camming.camPoints[point].SlaveAcc			:= -0.00195545;
_Camming.camPoints[point].SlaveJerk			:= 0.00;

//
point										:= 17;
_Camming.camPoints[point].MasterPos			:= 398.500;
_Camming.camPoints[point].SlavePos			:= 333.378;
_Camming.camPoints[point].PointIndex		:= point;
_Camming.camPoints[point].FunctionType		:= MC_MotionFunctionType.MOTIONFUNCTYPE_POLYNOM5_MM;
_Camming.camPoints[point].PointType			:= MC_MotionPointType.MOTIONPOINTTYPE_MOTION;
_Camming.camPoints[point].RelIndexNextPoint := 1;
_Camming.camPoints[point].SlaveVelo			:= 1.000000;
_Camming.camPoints[point].SlaveAcc			:= 0.00000000;
_Camming.camPoints[point].SlaveJerk			:= 0.00;

//
point										:= 18;
_Camming.camPoints[point].MasterPos			:= 666.600;
_Camming.camPoints[point].SlavePos			:= 601.478;
_Camming.camPoints[point].PointIndex		:= point;
_Camming.camPoints[point].FunctionType		:= MC_MotionFunctionType.MOTIONFUNCTYPE_POLYNOM5_MM;
_Camming.camPoints[point].PointType			:= MC_MotionPointType.MOTIONPOINTTYPE_MOTION;
_Camming.camPoints[point].RelIndexNextPoint := 1;
_Camming.camPoints[point].SlaveVelo			:= 1.000000;
_Camming.camPoints[point].SlaveAcc			:= 0.00000000;
_Camming.camPoints[point].SlaveJerk			:= 0.00;

//
point										:= 19;
_Camming.camPoints[point].MasterPos			:= 676.495;
_Camming.camPoints[point].SlavePos			:= 611.354;
_Camming.camPoints[point].PointIndex		:= point;
_Camming.camPoints[point].FunctionType		:= MC_MotionFunctionType.MOTIONFUNCTYPE_POLYNOM5_MM;
_Camming.camPoints[point].PointType			:= MC_MotionPointType.MOTIONPOINTTYPE_MOTION;
_Camming.camPoints[point].RelIndexNextPoint := 1;
_Camming.camPoints[point].SlaveVelo			:= 0.992814;
_Camming.camPoints[point].SlaveAcc			:= -0.00190944;
_Camming.camPoints[point].SlaveJerk			:= 0.00;

//
point										:= 20;
_Camming.camPoints[point].MasterPos			:= 686.390;
_Camming.camPoints[point].SlavePos			:= 621.030;
_Camming.camPoints[point].PointIndex		:= point;
_Camming.camPoints[point].FunctionType		:= MC_MotionFunctionType.MOTIONFUNCTYPE_POLYNOM5_MM;
_Camming.camPoints[point].PointType			:= MC_MotionPointType.MOTIONPOINTTYPE_MOTION;
_Camming.camPoints[point].RelIndexNextPoint := 1;
_Camming.camPoints[point].SlaveVelo			:= 0.957206;
_Camming.camPoints[point].SlaveAcc			:= -0.00535633;
_Camming.camPoints[point].SlaveJerk			:= 0.00;

//
point										:= 21;
_Camming.camPoints[point].MasterPos			:= 696.285;
_Camming.camPoints[point].SlavePos			:= 630.186;
_Camming.camPoints[point].PointIndex		:= point;
_Camming.camPoints[point].FunctionType		:= MC_MotionFunctionType.MOTIONFUNCTYPE_POLYNOM5_MM;
_Camming.camPoints[point].PointType			:= MC_MotionPointType.MOTIONPOINTTYPE_MOTION;
_Camming.camPoints[point].RelIndexNextPoint := 1;
_Camming.camPoints[point].SlaveVelo			:= 0.888425;
_Camming.camPoints[point].SlaveAcc			:= -0.00834680;
_Camming.camPoints[point].SlaveJerk			:= 0.00;

//
point										:= 22;
_Camming.camPoints[point].MasterPos			:= 706.180;
_Camming.camPoints[point].SlavePos			:= 638.538;
_Camming.camPoints[point].PointIndex		:= point;
_Camming.camPoints[point].FunctionType		:= MC_MotionFunctionType.MOTIONFUNCTYPE_POLYNOM5_MM;
_Camming.camPoints[point].PointType			:= MC_MotionPointType.MOTIONPOINTTYPE_MOTION;
_Camming.camPoints[point].RelIndexNextPoint := 1;
_Camming.camPoints[point].SlaveVelo			:= 0.797621;
_Camming.camPoints[point].SlaveAcc			:= -0.00966634;
_Camming.camPoints[point].SlaveJerk			:= 0.00;

//
point										:= 23;
_Camming.camPoints[point].MasterPos			:= 716.075;
_Camming.camPoints[point].SlavePos			:= 645.962;
_Camming.camPoints[point].PointIndex		:= point;
_Camming.camPoints[point].FunctionType		:= MC_MotionFunctionType.MOTIONFUNCTYPE_POLYNOM5_MM;
_Camming.camPoints[point].PointType			:= MC_MotionPointType.MOTIONPOINTTYPE_MOTION;
_Camming.camPoints[point].RelIndexNextPoint := 1;
_Camming.camPoints[point].SlaveVelo			:= 0.704244;
_Camming.camPoints[point].SlaveAcc			:= -0.00885381;
_Camming.camPoints[point].SlaveJerk			:= 0.00;

//
point										:= 24;
_Camming.camPoints[point].MasterPos			:= 725.970;
_Camming.camPoints[point].SlavePos			:= 652.534;
_Camming.camPoints[point].PointIndex		:= point;
_Camming.camPoints[point].FunctionType		:= MC_MotionFunctionType.MOTIONFUNCTYPE_POLYNOM5_MM;
_Camming.camPoints[point].PointType			:= MC_MotionPointType.MOTIONPOINTTYPE_MOTION;
_Camming.camPoints[point].RelIndexNextPoint := 1;
_Camming.camPoints[point].SlaveVelo			:= 0.628520;
_Camming.camPoints[point].SlaveAcc			:= -0.00621225;
_Camming.camPoints[point].SlaveJerk			:= 0.00;

//
point										:= 25;
_Camming.camPoints[point].MasterPos			:= 735.865;
_Camming.camPoints[point].SlavePos			:= 658.505;
_Camming.camPoints[point].PointIndex		:= point;
_Camming.camPoints[point].FunctionType		:= MC_MotionFunctionType.MOTIONFUNCTYPE_POLYNOM5_MM;
_Camming.camPoints[point].PointType			:= MC_MotionPointType.MOTIONPOINTTYPE_MOTION;
_Camming.camPoints[point].RelIndexNextPoint := 1;
_Camming.camPoints[point].SlaveVelo			:= 0.583944;
_Camming.camPoints[point].SlaveAcc			:= -0.00279152;
_Camming.camPoints[point].SlaveJerk			:= 0.00;

//
point										:= 26;
_Camming.camPoints[point].MasterPos			:= 745.760;
_Camming.camPoints[point].SlavePos			:= 664.195;
_Camming.camPoints[point].PointIndex		:= point;
_Camming.camPoints[point].FunctionType		:= MC_MotionFunctionType.MOTIONFUNCTYPE_POLYNOM5_MM;
_Camming.camPoints[point].PointType			:= MC_MotionPointType.MOTIONPOINTTYPE_MOTION;
_Camming.camPoints[point].RelIndexNextPoint := 1;
_Camming.camPoints[point].SlaveVelo			:= 0.570311;
_Camming.camPoints[point].SlaveAcc			:= -0.00028497;
_Camming.camPoints[point].SlaveJerk			:= 0.00;

//
point										:= 27;
_Camming.camPoints[point].MasterPos			:= 755.655;
_Camming.camPoints[point].SlavePos			:= 669.834;
_Camming.camPoints[point].PointIndex		:= point;
_Camming.camPoints[point].FunctionType		:= MC_MotionFunctionType.MOTIONFUNCTYPE_POLYNOM5_MM;
_Camming.camPoints[point].PointType			:= MC_MotionPointType.MOTIONPOINTTYPE_MOTION;
_Camming.camPoints[point].RelIndexNextPoint := 1;
_Camming.camPoints[point].SlaveVelo			:= 0.569785;
_Camming.camPoints[point].SlaveAcc			:= -0.00000641;
_Camming.camPoints[point].SlaveJerk			:= 0.00;

//
point										:= 28;
_Camming.camPoints[point].MasterPos			:= 765.550;
_Camming.camPoints[point].SlavePos			:= 675.476;
_Camming.camPoints[point].PointIndex		:= point;
_Camming.camPoints[point].FunctionType		:= MC_MotionFunctionType.MOTIONFUNCTYPE_POLYNOM5_MM;
_Camming.camPoints[point].PointType			:= MC_MotionPointType.MOTIONPOINTTYPE_MOTION;
_Camming.camPoints[point].RelIndexNextPoint := 1;
_Camming.camPoints[point].SlaveVelo			:= 0.571122;
_Camming.camPoints[point].SlaveAcc			:= 0.00033576;
_Camming.camPoints[point].SlaveJerk			:= 0.00;

//
point										:= 29;
_Camming.camPoints[point].MasterPos			:= 775.445;
_Camming.camPoints[point].SlavePos			:= 681.153;
_Camming.camPoints[point].PointIndex		:= point;
_Camming.camPoints[point].FunctionType		:= MC_MotionFunctionType.MOTIONFUNCTYPE_POLYNOM5_MM;
_Camming.camPoints[point].PointType			:= MC_MotionPointType.MOTIONPOINTTYPE_MOTION;
_Camming.camPoints[point].RelIndexNextPoint := 1;
_Camming.camPoints[point].SlaveVelo			:= 0.577454;
_Camming.camPoints[point].SlaveAcc			:= 0.00098723;
_Camming.camPoints[point].SlaveJerk			:= 0.00;

//
point										:= 30;
_Camming.camPoints[point].MasterPos			:= 785.340;
_Camming.camPoints[point].SlavePos			:= 686.929;
_Camming.camPoints[point].PointIndex		:= point;
_Camming.camPoints[point].FunctionType		:= MC_MotionFunctionType.MOTIONFUNCTYPE_POLYNOM5_MM;
_Camming.camPoints[point].PointType			:= MC_MotionPointType.MOTIONPOINTTYPE_MOTION;
_Camming.camPoints[point].RelIndexNextPoint := 1;
_Camming.camPoints[point].SlaveVelo			:= 0.591500;
_Camming.camPoints[point].SlaveAcc			:= 0.00188997;
_Camming.camPoints[point].SlaveJerk			:= 0.00;

//
point										:= 31;
_Camming.camPoints[point].MasterPos			:= 795.235;
_Camming.camPoints[point].SlavePos			:= 692.892;
_Camming.camPoints[point].PointIndex		:= point;
_Camming.camPoints[point].FunctionType		:= MC_MotionFunctionType.MOTIONFUNCTYPE_POLYNOM5_MM;
_Camming.camPoints[point].PointType			:= MC_MotionPointType.MOTIONPOINTTYPE_MOTION;
_Camming.camPoints[point].RelIndexNextPoint := 1;
_Camming.camPoints[point].SlaveVelo			:= 0.615664;
_Camming.camPoints[point].SlaveAcc			:= 0.00303751;
_Camming.camPoints[point].SlaveJerk			:= 0.00;

//
point										:= 32;
_Camming.camPoints[point].MasterPos			:= 805.130;
_Camming.camPoints[point].SlavePos			:= 699.155;
_Camming.camPoints[point].PointIndex		:= point;
_Camming.camPoints[point].FunctionType		:= MC_MotionFunctionType.MOTIONFUNCTYPE_POLYNOM5_MM;
_Camming.camPoints[point].PointType			:= MC_MotionPointType.MOTIONPOINTTYPE_MOTION;
_Camming.camPoints[point].RelIndexNextPoint := 1;
_Camming.camPoints[point].SlaveVelo			:= 0.652442;
_Camming.camPoints[point].SlaveAcc			:= 0.00443439;
_Camming.camPoints[point].SlaveJerk			:= 0.00;

//
point										:= 33;
_Camming.camPoints[point].MasterPos			:= 815.025;
_Camming.camPoints[point].SlavePos			:= 705.854;
_Camming.camPoints[point].PointIndex		:= point;
_Camming.camPoints[point].FunctionType		:= MC_MotionFunctionType.MOTIONFUNCTYPE_POLYNOM5_MM;
_Camming.camPoints[point].PointType			:= MC_MotionPointType.MOTIONPOINTTYPE_MOTION;
_Camming.camPoints[point].RelIndexNextPoint := 1;
_Camming.camPoints[point].SlaveVelo			:= 0.704402;
_Camming.camPoints[point].SlaveAcc			:= 0.00609093;
_Camming.camPoints[point].SlaveJerk			:= 0.00;

//
point										:= 34;
_Camming.camPoints[point].MasterPos			:= 824.920;
_Camming.camPoints[point].SlavePos			:= 713.150;
_Camming.camPoints[point].PointIndex		:= point;
_Camming.camPoints[point].FunctionType		:= MC_MotionFunctionType.MOTIONFUNCTYPE_POLYNOM5_MM;
_Camming.camPoints[point].PointType			:= MC_MotionPointType.MOTIONPOINTTYPE_MOTION;
_Camming.camPoints[point].RelIndexNextPoint := 1;
_Camming.camPoints[point].SlaveVelo			:= 0.773096;
_Camming.camPoints[point].SlaveAcc			:= 0.00774577;
_Camming.camPoints[point].SlaveJerk			:= 0.00;

//
point										:= 35;
_Camming.camPoints[point].MasterPos			:= 834.815;
_Camming.camPoints[point].SlavePos			:= 721.200;
_Camming.camPoints[point].PointIndex		:= point;
_Camming.camPoints[point].FunctionType		:= MC_MotionFunctionType.MOTIONFUNCTYPE_POLYNOM5_MM;
_Camming.camPoints[point].PointType			:= MC_MotionPointType.MOTIONPOINTTYPE_MOTION;
_Camming.camPoints[point].RelIndexNextPoint := 1;
_Camming.camPoints[point].SlaveVelo			:= 0.855433;
_Camming.camPoints[point].SlaveAcc			:= 0.00865192;
_Camming.camPoints[point].SlaveJerk			:= 0.00;

//
point										:= 36;
_Camming.camPoints[point].MasterPos			:= 844.710;
_Camming.camPoints[point].SlavePos			:= 730.077;
_Camming.camPoints[point].PointIndex		:= point;
_Camming.camPoints[point].FunctionType		:= MC_MotionFunctionType.MOTIONFUNCTYPE_POLYNOM5_MM;
_Camming.camPoints[point].PointType			:= MC_MotionPointType.MOTIONPOINTTYPE_MOTION;
_Camming.camPoints[point].RelIndexNextPoint := 1;
_Camming.camPoints[point].SlaveVelo			:= 0.936508;
_Camming.camPoints[point].SlaveAcc			:= 0.00721864;
_Camming.camPoints[point].SlaveJerk			:= 0.00;

//
point										:= 37;
_Camming.camPoints[point].MasterPos			:= 854.605;
_Camming.camPoints[point].SlavePos			:= 739.636;
_Camming.camPoints[point].PointIndex		:= point;
_Camming.camPoints[point].FunctionType		:= MC_MotionFunctionType.MOTIONFUNCTYPE_POLYNOM5_MM;
_Camming.camPoints[point].PointType			:= MC_MotionPointType.MOTIONPOINTTYPE_MOTION;
_Camming.camPoints[point].RelIndexNextPoint := 1;
_Camming.camPoints[point].SlaveVelo			:= 0.988558;
_Camming.camPoints[point].SlaveAcc			:= 0.00301892;
_Camming.camPoints[point].SlaveJerk			:= 0.00;

//
point										:= 38;
_Camming.camPoints[point].MasterPos			:= 864.500;
_Camming.camPoints[point].SlavePos			:= 749.500;
_Camming.camPoints[point].PointIndex		:= point;
_Camming.camPoints[point].FunctionType		:= MC_MotionFunctionType.MOTIONFUNCTYPE_POLYNOM5_MM;
_Camming.camPoints[point].PointType			:= MC_MotionPointType.MOTIONPOINTTYPE_MOTION;
_Camming.camPoints[point].RelIndexNextPoint := 1;
_Camming.camPoints[point].SlaveVelo			:= 1.000000;
_Camming.camPoints[point].SlaveAcc			:= 0.00000000;
_Camming.camPoints[point].SlaveJerk			:= 0.00;

//
point										:= 39;
_Camming.camPoints[point].MasterPos			:= 1000.500;
_Camming.camPoints[point].SlavePos			:= 885.500;
_Camming.camPoints[point].PointIndex		:= point;
_Camming.camPoints[point].FunctionType		:= MC_MotionFunctionType.MOTIONFUNCTYPE_POLYNOM5_MM;
_Camming.camPoints[point].PointType			:= MC_MotionPointType.MOTIONPOINTTYPE_MOTION;
_Camming.camPoints[point].RelIndexNextPoint := 1;
_Camming.camPoints[point].SlaveVelo			:= 1.000000;
_Camming.camPoints[point].SlaveAcc			:= 0.00000000;
_Camming.camPoints[point].SlaveJerk			:= 0.00;

//
point										:= 40;
_Camming.camPoints[point].MasterPos			:= 1010.367;
_Camming.camPoints[point].SlavePos			:= 895.398;
_Camming.camPoints[point].PointIndex		:= point;
_Camming.camPoints[point].FunctionType		:= MC_MotionFunctionType.MOTIONFUNCTYPE_POLYNOM5_MM;
_Camming.camPoints[point].PointType			:= MC_MotionPointType.MOTIONPOINTTYPE_MOTION;
_Camming.camPoints[point].RelIndexNextPoint := 1;
_Camming.camPoints[point].SlaveVelo			:= 1.011583;
_Camming.camPoints[point].SlaveAcc			:= 0.00312668;
_Camming.camPoints[point].SlaveJerk			:= 0.00;

//
point										:= 41;
_Camming.camPoints[point].MasterPos			:= 1020.233;
_Camming.camPoints[point].SlavePos			:= 905.622;
_Camming.camPoints[point].PointIndex		:= point;
_Camming.camPoints[point].FunctionType		:= MC_MotionFunctionType.MOTIONFUNCTYPE_POLYNOM5_MM;
_Camming.camPoints[point].PointType			:= MC_MotionPointType.MOTIONPOINTTYPE_MOTION;
_Camming.camPoints[point].RelIndexNextPoint := 1;
_Camming.camPoints[point].SlaveVelo			:= 1.070556;
_Camming.camPoints[point].SlaveAcc			:= 0.00898229;
_Camming.camPoints[point].SlaveJerk			:= 0.00;

